C09128=1014.857,84.775,382.125,166.252,57.206,160.405
C09129=1014.862,85.025,382.109,166.255,57.195,160.404
C09130=1014.867,85.274,382.093,166.257,57.185,160.402
C09131=1014.871,85.523,382.077,166.260,57.175,160.401
C09132=1014.876,85.772,382.061,166.262,57.164,160.399
C09133=1014.881,86.022,382.045,166.265,57.155,160.398
C09134=1014.886,86.271,382.028,166.267,57.144,160.397
C09135=1014.890,86.521,382.013,166.270,57.133,160.395
C09136=1014.895,86.771,381.996,166.272,57.124,160.394
C09137=1014.899,87.020,381.980,166.275,57.113,160.392
C09138=1014.904,87.269,381.963,166.277,57.102,160.391
C09139=1014.909,87.518,381.948,166.280,57.093,160.390
C09140=1014.914,87.768,381.931,166.282,57.082,160.388
C09141=1014.919,88.018,381.916,166.285,57.071,160.387
C09142=1014.923,88.267,381.899,166.288,57.061,160.386
C09143=1014.928,88.517,381.883,166.290,57.051,160.384
C09144=1014.933,88.766,381.866,166.292,57.041,160.382
C09145=1014.937,89.015,381.850,166.296,57.031,160.381
C09146=1014.942,89.265,381.834,166.297,57.020,160.380
C09147=1014.946,89.514,381.817,166.301,57.010,160.378
C09148=1014.951,89.763,381.800,166.302,57.000,160.377
C09149=1014.956,90.013,381.783,166.306,56.990,160.376
C09150=1014.960,90.294,381.766,166.309,56.978,160.374
C09151=1014.966,90.575,381.747,166.311,56.967,160.372
C09152=1014.970,90.855,381.728,166.314,56.955,160.371
C09153=1014.976,91.135,381.710,166.317,56.944,160.369
C09154=1014.980,91.384,381.693,166.319,56.934,160.368
C09155=1014.985,91.634,381.676,166.323,56.924,160.367
C09156=1014.990,91.884,381.660,166.324,56.914,160.365
C09157=1014.994,92.133,381.644,166.327,56.903,160.364
C09158=1015.000,92.382,381.627,166.330,56.893,160.363
C09159=1015.003,92.631,381.610,166.332,56.883,160.361
C09160=1015.008,92.880,381.593,166.335,56.872,160.360
C09161=1015.013,93.131,381.577,166.338,56.862,160.358
C09162=1015.018,93.380,381.560,166.340,56.852,160.357
C09163=1015.022,93.630,381.543,166.343,56.841,160.355
C09164=1015.027,93.879,381.527,166.346,56.831,160.354
C09165=1015.031,94.128,381.510,166.348,56.821,160.353
C09166=1015.036,94.378,381.494,166.350,56.811,160.351
C09167=1015.041,94.627,381.477,166.354,56.801,160.350
C09168=1015.045,94.876,381.460,166.355,56.790,160.348
C09169=1015.050,95.126,381.444,166.358,56.780,160.347
C09170=1015.055,95.375,381.427,166.361,56.770,160.346
C09171=1015.060,95.624,381.410,166.364,56.759,160.344
C09172=1015.064,95.873,381.394,166.366,56.749,160.343
C09173=1015.069,96.124,381.377,166.369,56.738,160.341
C09174=1015.073,96.373,381.360,166.372,56.728,160.340
C09175=1015.078,96.622,381.344,166.375,56.718,160.339
C09176=1015.083,96.871,381.327,166.376,56.708,160.337
C09177=1015.087,97.121,381.310,166.379,56.697,160.336
C09178=1015.092,97.370,381.293,166.382,56.686,160.334
C09179=1015.097,97.619,381.277,166.385,56.676,160.333
C09180=1015.102,97.869,381.260,166.387,56.666,160.332
C09181=1015.106,98.118,381.243,166.390,56.656,160.330
C09182=1015.110,98.367,381.226,166.393,56.645,160.329
C09183=1015.115,98.618,381.210,166.395,56.634,160.327
C09184=1015.120,98.866,381.194,166.399,56.625,160.326
C09185=1015.124,99.116,381.176,166.401,56.614,160.325
C09186=1015.129,99.365,381.159,166.403,56.604,160.323
C09187=1015.134,99.615,381.142,166.407,56.594,160.322
C09188=1015.138,99.864,381.125,166.408,56.584,160.320
C09189=1015.143,100.114,381.108,166.411,56.573,160.319
C09190=1015.147,100.363,381.091,166.415,56.563,160.318
C09191=1015.152,100.613,381.074,166.416,56.553,160.316
C09192=1015.157,100.862,381.057,166.419,56.542,160.315
C09193=1015.161,101.112,381.040,166.422,56.532,160.313
C09194=1015.166,101.360,381.023,166.424,56.522,160.312
C09195=1015.170,101.610,381.005,166.427,56.512,160.311
C09196=1015.175,101.859,380.989,166.430,56.501,160.309
C09197=1015.179,102.109,380.971,166.433,56.491,160.308
C09198=1015.184,102.358,380.955,166.435,56.481,160.307
C09199=1015.189,102.608,380.937,166.438,56.471,160.305
C09200=1015.193,102.857,380.921,166.441,56.460,160.304
C09201=1015.198,103.106,380.903,166.444,56.449,160.302
C09202=1015.203,103.355,380.886,166.446,56.440,160.301
C09203=1015.207,103.605,380.869,166.449,56.429,160.300
C09204=1015.212,103.854,380.852,166.452,56.419,160.298
C09205=1015.216,104.104,380.835,166.455,56.408,160.297
C09206=1015.221,104.352,380.818,166.457,56.399,160.296
C09207=1015.226,104.602,380.800,166.460,56.388,160.294
C09208=1015.229,104.851,380.783,166.463,56.378,160.293
C09209=1015.235,105.101,380.766,166.466,56.367,160.291
C09210=1015.239,105.350,380.748,166.467,56.357,160.290
C09211=1015.244,105.599,380.732,166.470,56.346,160.288
C09212=1015.248,105.849,380.714,166.474,56.336,160.287
C09213=1015.253,106.098,380.698,166.477,56.326,160.286
C09214=1015.259,106.379,380.678,166.480,56.314,160.284
C09215=1015.263,106.660,380.658,166.482,56.302,160.282
C09216=1015.269,106.940,380.639,166.485,56.290,160.281
C09217=1015.275,107.222,380.620,166.488,56.279,160.279
C09218=1015.279,107.471,380.602,166.491,56.268,160.278
C09219=1015.284,107.720,380.585,166.494,56.258,160.277
C09220=1015.288,107.970,380.568,166.498,56.248,160.275
C09221=1015.293,108.219,380.551,166.500,56.238,160.274
C09222=1015.298,108.469,380.533,166.502,56.227,160.272
C09223=1015.302,108.717,380.517,166.505,56.217,160.271
C09224=1015.307,108.967,380.499,166.508,56.206,160.270
C09225=1015.311,109.216,380.482,166.511,56.196,160.268
C09226=1015.316,109.466,380.465,166.514,56.185,160.267
C09227=1015.321,109.715,380.447,166.516,56.175,160.265
C09228=1015.325,109.964,380.430,166.519,56.164,160.264
C09229=1015.330,110.213,380.412,166.522,56.155,160.263
C09230=1015.335,110.463,380.395,166.525,56.144,160.261
C09231=1015.339,110.713,380.377,166.528,56.133,160.260
C09232=1015.344,110.962,380.359,166.530,56.123,160.258
C09233=1015.348,111.211,380.343,166.533,56.113,160.257
C09234=1015.353,111.460,380.325,166.536,56.102,160.256
C09235=1015.357,111.710,380.307,166.539,56.092,160.254
C09236=1015.362,111.959,380.289,166.542,56.081,160.253
C09237=1015.366,112.209,380.272,166.544,56.072,160.252
C09238=1015.371,112.458,380.254,166.547,56.061,160.250
C09239=1015.375,112.707,380.236,166.550,56.051,160.249
C09240=1015.380,112.957,380.219,166.553,56.040,160.247
C09241=1015.384,113.206,380.200,166.556,56.031,160.246
C09242=1015.389,113.455,380.183,166.558,56.020,160.245
C09243=1015.393,113.705,380.165,166.561,56.010,160.243
C09244=1015.398,113.954,380.147,166.564,55.999,160.242
C09245=1015.402,114.203,380.129,166.567,55.990,160.241
C09246=1015.406,114.453,380.112,166.570,55.980,160.239
C09247=1015.411,114.702,380.094,166.573,55.969,160.238
C09248=1015.415,114.951,380.076,166.576,55.959,160.237
C09249=1015.420,115.201,380.058,166.578,55.949,160.235
C09250=1015.425,115.450,380.040,166.581,55.939,160.234
C09251=1015.429,115.700,380.022,166.584,55.928,160.232
C09252=1015.434,115.948,380.004,166.587,55.918,160.231
C09253=1015.438,116.198,379.987,166.590,55.907,160.230
C09254=1015.443,116.447,379.969,166.592,55.897,160.228
C09255=1015.447,116.696,379.951,166.596,55.887,160.227
C09256=1015.452,116.945,379.933,166.599,55.877,160.226
C09257=1015.456,117.195,379.915,166.602,55.866,160.224
C09258=1015.460,117.416,379.900,166.604,55.857,160.223
C09259=1015.464,117.636,379.883,166.607,55.848,160.222
C09260=1015.469,117.857,379.867,166.610,55.839,160.221
C09261=1015.473,118.078,379.852,166.611,55.830,160.219
C09262=1015.477,118.298,379.836,166.614,55.821,160.218
C09263=1015.481,118.519,379.821,166.617,55.812,160.217
C09264=1015.484,118.740,379.804,166.619,55.803,160.216
C09265=1015.488,118.961,379.788,166.622,55.793,160.214
C09266=1015.493,119.210,379.770,166.625,55.783,160.213
C09267=1015.497,119.459,379.753,166.628,55.773,160.212
C09268=1015.502,119.708,379.734,166.631,55.762,160.210
C09269=1015.507,119.957,379.716,166.634,55.752,160.209
C09270=1015.512,120.207,379.698,166.636,55.742,160.208
C09271=1015.516,120.456,379.681,166.639,55.732,160.206
C09272=1015.520,120.705,379.663,166.642,55.721,160.205
C09273=1015.525,120.955,379.645,166.645,55.711,160.204
C09274=1015.530,121.204,379.626,166.648,55.700,160.202
C09275=1015.535,121.453,379.608,166.651,55.690,160.201
C09276=1015.539,121.702,379.591,166.654,55.680,160.199
C09277=1015.543,121.952,379.573,166.657,55.669,160.198
C09278=1015.550,122.290,379.548,166.660,55.655,160.196
C09279=1015.556,122.628,379.524,166.665,55.641,160.194
C09280=1015.563,122.967,379.499,166.669,55.627,160.192
C09281=1015.568,123.305,379.475,166.674,55.613,160.191
C09282=1015.573,123.554,379.457,166.677,55.602,160.189
C09283=1015.578,123.804,379.439,166.680,55.592,160.188
C09284=1015.583,124.053,379.420,166.682,55.582,160.186
C09285=1015.588,124.302,379.402,166.685,55.571,160.185
C09286=1015.592,124.551,379.384,166.688,55.561,160.184
C09287=1015.597,124.800,379.366,166.691,55.551,160.182
C09288=1015.601,125.050,379.348,166.694,55.540,160.181
C09289=1015.606,125.299,379.330,166.697,55.530,160.180
C09290=1015.611,125.549,379.313,166.700,55.519,160.178
C09291=1015.615,125.798,379.294,166.703,55.509,160.177
C09292=1015.620,126.048,379.276,166.706,55.498,160.175
C09293=1015.625,126.297,379.258,166.709,55.487,160.174
C09294=1015.629,126.546,379.240,166.712,55.477,160.173
C09295=1015.634,126.795,379.222,166.715,55.466,160.171
C09296=1015.639,127.044,379.204,166.718,55.456,160.170
C09297=1015.643,127.294,379.186,166.722,55.446,160.168
C09298=1015.648,127.543,379.168,166.725,55.435,160.167
C09299=1015.653,127.792,379.149,166.728,55.425,160.166
C09300=1015.658,128.042,379.131,166.731,55.414,160.164
C09301=1015.663,128.291,379.113,166.734,55.404,160.163
C09302=1015.667,128.540,379.095,166.737,55.394,160.162
C09303=1015.671,128.790,379.076,166.740,55.383,160.160
C09304=1015.676,129.039,379.057,166.743,55.372,160.159
C09305=1015.681,129.288,379.039,166.746,55.362,160.157
C09306=1015.685,129.537,379.021,166.749,55.351,160.156
C09307=1015.690,129.786,379.003,166.752,55.341,160.155
C09308=1015.694,130.036,378.984,166.755,55.330,160.153
C09309=1015.700,130.286,378.966,166.758,55.320,160.152
C09310=1015.704,130.535,378.948,166.762,55.310,160.151
C09311=1015.708,130.784,378.929,166.765,55.300,160.149
C09312=1015.713,131.033,378.911,166.768,55.290,160.148
C09313=1015.717,131.283,378.892,166.772,55.279,160.147
C09314=1015.722,131.531,378.873,166.775,55.269,160.145
C09315=1015.727,131.781,378.855,166.777,55.259,160.144
C09316=1015.731,132.030,378.836,166.780,55.249,160.143
C09317=1015.736,132.280,378.818,166.783,55.238,160.141
C09318=1015.740,132.529,378.798,166.786,55.228,160.140
C09319=1015.745,132.778,378.780,166.789,55.217,160.138
C09320=1015.750,133.027,378.762,166.793,55.207,160.137
C09321=1015.754,133.276,378.743,166.796,55.197,160.136
C09322=1015.759,133.526,378.724,166.799,55.186,160.134
C09323=1015.763,133.775,378.706,166.802,55.176,160.133
C09324=1015.768,134.024,378.687,166.805,55.166,160.132
C09325=1015.773,134.274,378.669,166.808,55.155,160.130
C09326=1015.777,134.523,378.650,166.812,55.145,160.129
C09327=1015.782,134.772,378.631,166.815,55.135,160.128
C09328=1015.786,135.021,378.613,166.818,55.124,160.126
C09329=1015.791,135.270,378.593,166.821,55.114,160.125
C09330=1015.796,135.520,378.575,166.824,55.103,160.124
C09331=1015.800,135.769,378.556,166.828,55.093,160.122
C09332=1015.805,136.018,378.538,166.831,55.083,160.121
C09333=1015.809,136.268,378.519,166.834,55.072,160.120
C09334=1015.814,136.516,378.500,166.837,55.062,160.118
C09335=1015.818,136.766,378.481,166.840,55.052,160.117
C09336=1015.823,137.015,378.462,166.844,55.041,160.116
C09337=1015.828,137.265,378.443,166.847,55.031,160.114
C09338=1015.833,137.514,378.424,166.850,55.021,160.113
C09339=1015.837,137.764,378.406,166.853,55.010,160.112
C09340=1015.842,138.012,378.387,166.856,55.000,160.110
C09341=1015.846,138.262,378.368,166.860,54.990,160.109
C09342=1015.851,138.543,378.346,166.863,54.978,160.107
C09343=1015.856,138.823,378.325,166.867,54.967,160.106
C09344=1015.861,139.104,378.304,166.871,54.955,160.105
C09345=1015.866,139.385,378.282,166.874,54.943,160.103
C09346=1015.871,139.634,378.263,166.877,54.933,160.102
C09347=1015.875,139.884,378.244,166.881,54.923,160.100
C09348=1015.879,140.133,378.225,166.884,54.913,160.099
C09349=1015.885,140.382,378.205,166.888,54.903,160.098
C09350=1015.889,140.632,378.187,166.891,54.892,160.096
C09351=1015.894,140.881,378.167,166.894,54.882,160.095
C09352=1015.899,141.129,378.148,166.897,54.872,160.094
C09353=1015.903,141.379,378.130,166.901,54.861,160.092
C09354=1015.907,141.628,378.110,166.904,54.851,160.091
C09355=1015.912,141.877,378.091,166.907,54.841,160.090
C09356=1015.916,142.127,378.072,166.910,54.831,160.088
C09357=1015.921,142.376,378.053,166.914,54.820,160.087
C09358=1015.926,142.625,378.034,166.917,54.810,160.086
C09359=1015.930,142.875,378.015,166.920,54.800,160.084
C09360=1015.935,143.123,377.996,166.923,54.789,160.083
C09361=1015.940,143.373,377.977,166.927,54.779,160.082
C09362=1015.944,143.622,377.957,166.930,54.769,160.080
C09363=1015.949,143.872,377.939,166.933,54.759,160.079
C09364=1015.954,144.121,377.919,166.937,54.748,160.078
C09365=1015.958,144.370,377.900,166.940,54.738,160.076
C09366=1015.963,144.618,377.881,166.943,54.728,160.075
C09367=1015.967,144.868,377.862,166.946,54.717,160.074
C09368=1015.972,145.117,377.843,166.950,54.707,160.072
C09369=1015.977,145.367,377.823,166.953,54.697,160.071
C09370=1015.982,145.616,377.804,166.956,54.687,160.070
C09371=1015.986,145.865,377.784,166.960,54.676,160.068
C09372=1015.990,146.114,377.765,166.963,54.666,160.067
C09373=1015.995,146.363,377.745,166.966,54.656,160.066
C09374=1015.999,146.613,377.726,166.970,54.645,160.064
C09375=1016.004,146.862,377.707,166.973,54.635,160.063
C09376=1016.008,147.111,377.687,166.976,54.625,160.062
C09377=1016.013,147.360,377.669,166.979,54.615,160.061
C09378=1016.018,147.610,377.649,166.984,54.604,160.059
C09379=1016.022,147.859,377.629,166.987,54.594,160.058
C09380=1016.027,148.108,377.610,166.990,54.583,160.057
C09381=1016.031,148.357,377.590,166.994,54.573,160.055
C09382=1016.036,148.607,377.570,166.997,54.563,160.054
C09383=1016.040,148.856,377.551,167.000,54.553,160.053
C09384=1016.045,149.105,377.531,167.004,54.543,160.052
C09385=1016.049,149.354,377.512,167.008,54.533,160.050
C09386=1016.054,149.603,377.492,167.011,54.523,160.049
C09387=1016.058,149.852,377.473,167.014,54.512,160.048
C09388=1016.063,150.101,377.453,167.018,54.502,160.046
C09389=1016.068,150.351,377.433,167.021,54.492,160.045
C09390=1016.072,150.600,377.414,167.024,54.482,160.044
C09391=1016.077,150.849,377.395,167.028,54.472,160.042
C09392=1016.082,151.097,377.375,167.031,54.461,160.041
C09393=1016.087,151.347,377.355,167.034,54.451,160.040
C09394=1016.091,151.596,377.336,167.038,54.441,160.038
C09395=1016.095,151.845,377.316,167.041,54.431,160.037
C09396=1016.100,152.095,377.296,167.045,54.420,160.036
C09397=1016.105,152.344,377.277,167.049,54.410,160.035
C09398=1016.109,152.593,377.257,167.052,54.400,160.033
C09399=1016.114,152.843,377.237,167.056,54.389,160.032
C09400=1016.119,153.091,377.217,167.059,54.379,160.031
C09401=1016.123,153.340,377.198,167.062,54.369,160.029
C09402=1016.127,153.590,377.177,167.066,54.359,160.028
C09403=1016.132,153.839,377.158,167.070,54.349,160.027
C09404=1016.136,154.088,377.138,167.073,54.339,160.026
C09405=1016.141,154.338,377.118,167.076,54.329,160.024
C09406=1016.146,154.618,377.096,167.080,54.317,160.023
C09407=1016.152,154.899,377.073,167.084,54.305,160.021
C09408=1016.157,155.180,377.051,167.089,54.294,160.020
C09409=1016.162,155.460,377.029,167.093,54.282,160.019
C09410=1016.166,155.710,377.008,167.096,54.272,160.017
C09411=1016.171,155.959,376.989,167.099,54.262,160.016
C09412=1016.176,156.209,376.969,167.103,54.252,160.015
C09413=1016.180,156.457,376.949,167.106,54.242,160.013
C09414=1016.185,156.706,376.929,167.110,54.231,160.012
C09415=1016.189,156.956,376.909,167.113,54.221,160.011
C09416=1016.194,157.204,376.889,167.118,54.211,160.010
C09417=1016.199,157.454,376.869,167.121,54.201,160.008
C09418=1016.203,157.703,376.850,167.125,54.191,160.007
C09419=1016.207,157.952,376.829,167.128,54.181,160.006
C09420=1016.212,158.202,376.809,167.132,54.171,160.004
C09421=1016.217,158.451,376.790,167.135,54.160,160.003
C09422=1016.222,158.700,376.769,167.139,54.150,160.002
C09423=1016.226,158.948,376.749,167.142,54.140,160.001
C09424=1016.231,159.198,376.729,167.146,54.131,159.999
C09425=1016.235,159.447,376.708,167.149,54.121,159.998
C09426=1016.238,159.696,376.688,167.153,54.110,159.997
C09427=1016.244,159.945,376.667,167.157,54.101,159.996
C09428=1016.247,160.194,376.646,167.160,54.091,159.994
C09429=1016.252,160.444,376.627,167.164,54.081,159.993
C09430=1016.256,160.693,376.606,167.167,54.070,159.992
C09431=1016.261,160.942,376.585,167.171,54.061,159.991
C09432=1016.265,161.191,376.565,167.174,54.051,159.990
C09433=1016.270,161.441,376.544,167.178,54.041,159.988
C09434=1016.274,161.689,376.524,167.181,54.030,159.987
C09435=1016.279,161.938,376.503,167.185,54.021,159.986
C09436=1016.283,162.187,376.483,167.190,54.010,159.985
C09437=1016.287,162.436,376.463,167.193,54.000,159.983
C09438=1016.292,162.686,376.441,167.197,53.991,159.982
C09439=1016.296,162.935,376.422,167.201,53.981,159.981
C09440=1016.301,163.184,376.401,167.204,53.971,159.980
C09441=1016.306,163.433,376.380,167.208,53.960,159.978
C09442=1016.310,163.682,376.359,167.211,53.951,159.977
C09443=1016.314,163.932,376.339,167.215,53.941,159.976
C09444=1016.319,164.180,376.319,167.218,53.931,159.975
C09445=1016.323,164.430,376.298,167.222,53.921,159.973
C09446=1016.328,164.678,376.277,167.226,53.911,159.972
C09447=1016.332,164.928,376.256,167.229,53.901,159.971
C09448=1016.337,165.177,376.237,167.234,53.891,159.970
C09449=1016.341,165.426,376.216,167.237,53.880,159.969
C09450=1016.345,165.675,376.195,167.241,53.870,159.967
C09451=1016.350,165.924,376.174,167.245,53.861,159.966
C09452=1016.354,166.173,376.154,167.248,53.851,159.965
C09453=1016.359,166.422,376.133,167.252,53.841,159.964
C09454=1016.364,166.672,376.113,167.255,53.831,159.962
C09455=1016.368,166.921,376.092,167.259,53.821,159.961
C09456=1016.373,167.170,376.071,167.264,53.811,159.960
C09457=1016.377,167.419,376.050,167.267,53.801,159.959
C09458=1016.382,167.668,376.030,167.271,53.790,159.957
C09459=1016.387,167.917,376.009,167.274,53.780,159.956
C09460=1016.390,168.166,375.988,167.278,53.771,159.955
C09461=1016.396,168.415,375.967,167.282,53.761,159.954
C09462=1016.400,168.664,375.946,167.286,53.750,159.953
C09463=1016.405,168.913,375.926,167.290,53.740,159.951
C09464=1016.409,169.163,375.906,167.294,53.730,159.950
C09465=1016.413,169.412,375.885,167.298,53.721,159.949
C09466=1016.418,169.661,375.864,167.301,53.711,159.948
C09467=1016.423,169.910,375.843,167.306,53.700,159.947
C09468=1016.427,170.159,375.823,167.309,53.690,159.945
C09469=1016.432,170.408,375.802,167.313,53.680,159.944
C09470=1016.437,170.688,375.778,167.317,53.669,159.943
C09471=1016.443,170.969,375.755,167.321,53.658,159.941
C09472=1016.447,171.250,375.732,167.326,53.646,159.940
C09473=1016.453,171.530,375.707,167.330,53.635,159.938
C09474=1016.458,171.779,375.687,167.334,53.625,159.937
C09475=1016.462,172.028,375.666,167.339,53.615,159.936
C09476=1016.467,172.277,375.645,167.342,53.605,159.935
C09477=1016.472,172.527,375.624,167.346,53.595,159.934
C09478=1016.476,172.775,375.603,167.349,53.585,159.932
C09479=1016.481,173.024,375.583,167.354,53.575,159.931
C09480=1016.486,173.274,375.562,167.358,53.564,159.930
C09481=1016.490,173.522,375.542,167.362,53.555,159.929
C09482=1016.495,173.772,375.520,167.365,53.545,159.928
C09483=1016.499,174.021,375.499,167.370,53.535,159.926
C09484=1016.505,174.270,375.479,167.373,53.525,159.925
C09485=1016.509,174.520,375.458,167.377,53.515,159.924
C09486=1016.513,174.769,375.437,167.382,53.505,159.923
C09487=1016.519,175.017,375.416,167.386,53.495,159.922
C09488=1016.523,175.266,375.394,167.389,53.485,159.920
C09489=1016.528,175.516,375.374,167.393,53.475,159.919
C09490=1016.532,175.764,375.353,167.397,53.464,159.918
C09491=1016.537,176.014,375.332,167.401,53.454,159.917
C09492=1016.542,176.263,375.311,167.405,53.444,159.915
C09493=1016.547,176.512,375.289,167.410,53.434,159.914
C09494=1016.552,176.761,375.269,167.413,53.424,159.913
C09495=1016.557,177.010,375.248,167.417,53.414,159.912
C09496=1016.561,177.259,375.227,167.422,53.404,159.911
C09497=1016.566,177.508,375.206,167.425,53.394,159.909
C09498=1016.571,177.757,375.185,167.429,53.384,159.908
C09499=1016.576,178.006,375.164,167.434,53.374,159.907
C09500=1016.580,178.255,375.143,167.438,53.364,159.906
C09501=1016.585,178.505,375.122,167.442,53.354,159.905
C09502=1016.590,178.753,375.100,167.446,53.344,159.903
C09503=1016.594,179.002,375.080,167.449,53.334,159.902
C09504=1016.599,179.252,375.059,167.454,53.323,159.901
C09505=1016.604,179.501,375.038,167.458,53.313,159.900
C09506=1016.609,179.750,375.016,167.462,53.304,159.899
C09507=1016.614,179.999,374.996,167.466,53.294,159.897
C09508=1016.619,180.248,374.974,167.470,53.284,159.896
C09509=1016.624,180.497,374.953,167.475,53.273,159.895
C09510=1016.629,180.746,374.932,167.478,53.263,159.894
C09511=1016.633,180.995,374.911,167.482,53.253,159.892
C09512=1016.638,181.244,374.889,167.487,53.244,159.891
C09513=1016.643,181.493,374.868,167.491,53.234,159.890
C09514=1016.648,181.742,374.847,167.495,53.223,159.889
C09515=1016.653,181.992,374.825,167.499,53.213,159.888
C09516=1016.658,182.240,374.804,167.503,53.204,159.887
C09517=1016.661,182.490,374.782,167.507,53.194,159.885
C09518=1016.666,182.738,374.760,167.512,53.184,159.884
C09519=1016.670,182.987,374.738,167.516,53.174,159.883
C09520=1016.674,183.237,374.717,167.520,53.165,159.882
C09521=1016.679,183.486,374.695,167.523,53.155,159.881
C09522=1016.684,183.735,374.673,167.529,53.145,159.880
C09523=1016.689,183.983,374.651,167.532,53.135,159.879
C09524=1016.693,184.232,374.629,167.536,53.126,159.878
C09525=1016.697,184.482,374.607,167.540,53.116,159.876
C09526=1016.702,184.731,374.586,167.545,53.106,159.875
C09527=1016.707,184.980,374.564,167.549,53.097,159.874
C09528=1016.711,185.229,374.541,167.553,53.087,159.873
C09529=1016.716,185.477,374.519,167.557,53.077,159.872
C09530=1016.720,185.727,374.498,167.561,53.067,159.871
C09531=1016.724,185.976,374.476,167.566,53.058,159.869
C09532=1016.729,186.225,374.454,167.569,53.048,159.868
C09533=1016.734,186.474,374.432,167.574,53.038,159.867
C09534=1016.739,186.754,374.408,167.579,53.027,159.866
C09535=1016.744,187.034,374.382,167.583,53.016,159.865
C09536=1016.750,187.315,374.358,167.589,53.005,159.863
C09537=1016.754,187.594,374.333,167.593,52.994,159.862
C09538=1016.759,187.844,374.312,167.597,52.984,159.861
C09539=1016.764,188.093,374.290,167.602,52.975,159.860
C09540=1016.768,188.341,374.268,167.606,52.965,159.859
C09541=1016.772,188.590,374.246,167.610,52.956,159.858
C09542=1016.778,188.840,374.223,167.614,52.945,159.856
C09543=1016.783,189.089,374.201,167.619,52.936,159.855
C09544=1016.787,189.338,374.180,167.623,52.926,159.854
C09545=1016.792,189.587,374.157,167.628,52.916,159.853
C09546=1016.796,189.836,374.135,167.631,52.907,159.852
C09547=1016.801,190.084,374.113,167.636,52.897,159.851
C09548=1016.805,190.333,374.091,167.640,52.887,159.850
C09549=1016.810,190.582,374.069,167.644,52.878,159.849
C09550=1016.815,190.831,374.047,167.649,52.867,159.847
C09551=1016.820,191.080,374.025,167.653,52.858,159.846
C09552=1016.824,191.330,374.003,167.658,52.848,159.845
C09553=1016.829,191.579,373.981,167.662,52.839,159.844
C09554=1016.834,191.827,373.959,167.666,52.829,159.843
C09555=1016.838,192.077,373.936,167.671,52.819,159.842
C09556=1016.843,192.325,373.914,167.675,52.809,159.841
C09557=1016.848,192.574,373.893,167.680,52.799,159.840
C09558=1016.854,192.823,373.870,167.684,52.790,159.838
C09559=1016.858,193.072,373.847,167.689,52.780,159.837
C09560=1016.862,193.321,373.825,167.693,52.770,159.836
C09561=1016.867,193.570,373.803,167.698,52.760,159.835
C09562=1016.871,193.819,373.781,167.702,52.751,159.834
C09563=1016.877,194.068,373.759,167.706,52.741,159.833
C09564=1016.882,194.317,373.737,167.711,52.731,159.832
C09565=1016.886,194.566,373.714,167.715,52.722,159.831
C09566=1016.891,194.815,373.692,167.720,52.712,159.830
C09567=1016.896,195.063,373.670,167.724,52.702,159.828
C09568=1016.901,195.313,373.648,167.729,52.693,159.827
C09569=1016.905,195.562,373.625,167.733,52.683,159.826
C09570=1016.910,195.811,373.603,167.738,52.673,159.825
C09571=1016.915,196.059,373.581,167.742,52.663,159.824
C09572=1016.920,196.309,373.558,167.747,52.654,159.823
C09573=1016.925,196.558,373.536,167.751,52.644,159.822
C09574=1016.929,196.806,373.514,167.756,52.634,159.821
C09575=1016.934,197.056,373.491,167.760,52.624,159.819
C09576=1016.939,197.305,373.469,167.765,52.615,159.819
C09577=1016.944,197.553,373.447,167.769,52.605,159.817
C09578=1016.950,197.802,373.424,167.774,52.595,159.816
C09579=1016.954,198.051,373.402,167.779,52.585,159.815
C09580=1016.959,198.300,373.380,167.783,52.576,159.814
C09581=1016.964,198.549,373.357,167.788,52.566,159.813
C09582=1016.969,198.798,373.334,167.792,52.556,159.812
C09583=1016.973,199.047,373.313,167.797,52.546,159.811
C09584=1016.979,199.296,373.290,167.801,52.537,159.810
C09585=1016.983,199.545,373.267,167.806,52.527,159.809
C09586=1016.988,199.794,373.244,167.810,52.518,159.808
C09587=1016.992,200.043,373.221,167.816,52.508,159.807
C09588=1016.997,200.292,373.199,167.819,52.499,159.805
C09589=1017.002,200.541,373.176,167.825,52.489,159.804
C09590=1017.006,200.790,373.153,167.829,52.480,159.803
C09591=1017.012,201.038,373.130,167.834,52.470,159.802
C09592=1017.016,201.287,373.108,167.838,52.460,159.801
C09593=1017.021,201.536,373.084,167.843,52.451,159.800
C09594=1017.026,201.785,373.061,167.847,52.441,159.799
C09595=1017.030,202.033,373.038,167.852,52.432,159.798
C09596=1017.035,202.281,373.016,167.857,52.423,159.797
C09597=1017.058,203.524,372.902,168.348,52.501,159.911
C09598=1017.064,203.761,372.878,168.352,52.493,159.910
C09599=1017.070,203.999,372.855,168.356,52.485,159.909
C09600=1017.075,204.236,372.832,168.359,52.477,159.908
C09601=1017.081,204.474,372.808,168.364,52.469,159.907
C09602=1017.086,204.712,372.785,168.368,52.461,159.906
C09603=1017.092,204.949,372.761,168.371,52.453,159.905
C09604=1017.097,205.187,372.737,168.375,52.445,159.904
C09605=1017.103,205.425,372.714,168.379,52.437,159.903
C09606=1017.109,205.673,372.689,168.383,52.429,159.902
C09607=1017.114,205.922,372.665,168.387,52.421,159.901
C09608=1017.120,206.171,372.640,168.390,52.413,159.900
C09609=1017.126,206.419,372.615,168.395,52.404,159.899
C09610=1017.132,206.668,372.590,168.399,52.396,159.898
C09611=1017.138,206.916,372.566,168.403,52.387,159.897
C09612=1017.144,207.165,372.541,168.407,52.379,159.896
C09613=1017.149,207.413,372.516,168.411,52.371,159.895
C09614=1017.155,207.663,372.491,168.415,52.362,159.894
C09615=1017.160,207.912,372.467,168.418,52.354,159.893
C09616=1017.166,208.160,372.442,168.423,52.346,159.892
C09617=1017.172,208.409,372.417,168.427,52.338,159.891
C09618=1017.178,208.657,372.392,168.431,52.330,159.890
C09619=1017.183,208.907,372.367,168.435,52.322,159.889
C09620=1017.189,209.155,372.342,168.439,52.314,159.888
C09621=1017.195,209.404,372.318,168.444,52.306,159.888
C09622=1017.201,209.653,372.292,168.447,52.298,159.887
C09623=1017.207,209.901,372.268,168.451,52.290,159.886
C09624=1017.212,210.150,372.242,168.456,52.281,159.885
C09625=1017.218,210.398,372.217,168.459,52.273,159.884
C09626=1017.224,210.647,372.192,168.463,52.265,159.883
C09627=1017.230,210.896,372.167,168.468,52.258,159.882
C09628=1017.235,211.144,372.142,168.472,52.250,159.881
C09629=1017.241,211.393,372.116,168.475,52.242,159.880
C09630=1017.246,211.642,372.092,168.479,52.234,159.879
C09631=1017.252,211.890,372.067,168.484,52.226,159.878
C09632=1017.258,212.139,372.041,168.488,52.218,159.877
C09633=1017.263,212.388,372.017,168.491,52.210,159.876
C09634=1017.269,212.636,371.991,168.496,52.202,159.875
C09635=1017.275,212.885,371.966,168.500,52.194,159.875
C09636=1017.280,213.133,371.940,168.504,52.186,159.874
C09637=1017.286,213.383,371.916,168.507,52.178,159.873
C09638=1017.292,213.631,371.890,168.513,52.171,159.872
C09639=1017.298,213.879,371.866,168.516,52.163,159.871
C09640=1017.303,214.128,371.840,168.520,52.155,159.870
C09641=1017.310,214.377,371.814,168.524,52.147,159.869
C09642=1017.316,214.626,371.790,168.529,52.139,159.868
C09643=1017.321,214.874,371.765,168.533,52.132,159.867
C09644=1017.327,215.123,371.739,168.536,52.124,159.866
C09645=1017.333,215.372,371.713,168.540,52.116,159.865
C09646=1017.338,215.620,371.688,168.545,52.108,159.865
C09647=1017.345,215.869,371.663,168.549,52.100,159.864
C09648=1017.350,216.118,371.638,168.553,52.093,159.863
C09649=1017.356,216.367,371.613,168.557,52.085,159.862
C09650=1017.362,216.615,371.588,168.562,52.077,159.861
C09651=1017.367,216.864,371.562,168.565,52.069,159.860
C09652=1017.373,217.112,371.536,168.570,52.062,159.859
C09653=1017.379,217.361,371.511,168.573,52.054,159.858
C09654=1017.385,217.609,371.486,168.578,52.046,159.858
C09655=1017.391,217.858,371.460,168.582,52.038,159.857
C09656=1017.397,218.107,371.435,168.586,52.031,159.856
C09657=1017.403,218.355,371.409,168.590,52.023,159.855
C09658=1017.408,218.590,371.385,168.594,52.016,159.854
C09659=1017.414,218.824,371.361,168.598,52.008,159.853
C09660=1017.419,219.059,371.337,168.602,52.002,159.853
C09661=1017.424,219.294,371.313,168.606,51.995,159.852
C09662=1017.429,219.528,371.288,168.610,51.987,159.851
C09663=1017.434,219.763,371.263,168.613,51.980,159.850
C09664=1017.440,219.998,371.240,168.617,51.973,159.849
C09665=1017.445,220.233,371.215,168.621,51.966,159.849
C09666=1017.451,220.481,371.190,168.625,51.959,159.848
C09667=1017.457,220.729,371.163,168.629,51.951,159.847
C09668=1017.463,220.978,371.138,168.634,51.944,159.846
C09669=1017.469,221.227,371.112,168.637,51.936,159.845
C09670=1017.475,221.476,371.087,168.641,51.929,159.844
C09671=1017.480,221.724,371.061,168.647,51.921,159.844
C09672=1017.487,221.973,371.035,168.651,51.914,159.843
C09673=1017.492,222.221,371.009,168.655,51.907,159.842
C09674=1017.497,222.470,370.983,168.659,51.899,159.841
C09675=1017.503,222.718,370.958,168.663,51.891,159.840
C09676=1017.509,222.967,370.931,168.667,51.884,159.840
C09677=1017.515,223.215,370.906,168.671,51.877,159.839
C09678=1017.521,223.464,370.880,168.675,51.870,159.838
C09679=1017.527,223.713,370.855,168.679,51.862,159.837
C09680=1017.533,223.961,370.828,168.683,51.855,159.836
C09681=1017.538,224.210,370.802,168.687,51.848,159.836
C09682=1017.544,224.459,370.777,168.692,51.841,159.835
C09683=1017.550,224.708,370.750,168.697,51.833,159.834
C09684=1017.556,224.956,370.725,168.701,51.826,159.833
C09685=1017.561,225.204,370.699,168.705,51.818,159.833
C09686=1017.567,225.453,370.673,168.709,51.811,159.831
C09687=1017.573,225.701,370.647,168.713,51.803,159.831
C09688=1017.579,225.950,370.621,168.717,51.796,159.830
C09689=1017.585,226.199,370.595,168.721,51.789,159.829
C09690=1017.591,226.447,370.569,168.725,51.782,159.828
C09691=1017.596,226.696,370.543,168.730,51.775,159.828
C09692=1017.603,226.944,370.517,168.734,51.768,159.827
C09693=1017.608,227.193,370.491,168.738,51.760,159.826
C09694=1017.614,227.441,370.464,168.742,51.753,159.825
C09695=1017.620,227.690,370.438,168.747,51.746,159.825
C09696=1017.625,227.939,370.411,168.751,51.739,159.824
C09697=1017.631,228.188,370.386,168.755,51.732,159.823
C09698=1017.637,228.436,370.359,168.759,51.725,159.822
C09699=1017.643,228.684,370.333,168.764,51.718,159.822
C09700=1017.649,228.933,370.307,168.768,51.710,159.821
C09701=1017.654,229.181,370.280,168.772,51.704,159.820
C09702=1017.660,229.430,370.254,168.776,51.697,159.819
C09703=1017.666,229.679,370.228,168.781,51.689,159.819
C09704=1017.672,229.927,370.202,168.785,51.682,159.818
C09705=1017.678,230.175,370.175,168.788,51.676,159.817
C09706=1017.683,230.424,370.149,168.793,51.669,159.816
C09707=1017.690,230.673,370.122,168.797,51.662,159.816
C09708=1017.696,230.921,370.095,168.801,51.655,159.815
C09709=1017.701,231.170,370.069,168.805,51.648,159.814
C09710=1017.707,231.419,370.043,168.810,51.641,159.814
C09711=1017.713,231.667,370.016,168.814,51.634,159.813
C09712=1017.718,231.916,369.990,168.818,51.627,159.812
C09713=1017.724,232.164,369.963,168.823,51.620,159.812
C09714=1017.730,232.412,369.936,168.827,51.613,159.811
C09715=1017.736,232.661,369.910,168.832,51.606,159.810
C09716=1017.741,232.910,369.884,168.835,51.600,159.809
C09717=1017.747,233.159,369.857,168.840,51.593,159.809
C09718=1017.752,233.389,369.832,168.844,51.586,159.808
C09719=1017.758,233.619,369.807,168.848,51.580,159.807
C09720=1017.764,233.850,369.783,168.851,51.574,159.807
C09721=1017.769,234.080,369.758,168.856,51.568,159.806
C09722=1017.774,234.310,369.733,168.859,51.561,159.805
C09723=1017.780,234.542,369.709,168.864,51.555,159.805
C09724=1017.785,234.772,369.684,168.868,51.549,159.804
C09725=1017.790,235.002,369.659,168.871,51.543,159.804
C09726=1017.797,235.251,369.632,168.875,51.535,159.803
C09727=1017.802,235.499,369.605,168.880,51.529,159.802
C09728=1017.808,235.748,369.579,168.884,51.522,159.801
C09729=1017.814,235.996,369.552,168.889,51.515,159.801
C09730=1017.820,236.244,369.525,168.893,51.509,159.800
C09731=1017.826,236.493,369.498,168.898,51.501,159.799
C09732=1017.832,236.742,369.472,168.901,51.495,159.799
C09733=1017.838,236.990,369.445,168.906,51.489,159.798
C09734=1017.843,237.238,369.418,168.910,51.481,159.797
C09735=1017.850,237.488,369.391,168.915,51.475,159.797
C09736=1017.856,237.736,369.365,168.919,51.468,159.796
C09737=1017.861,237.984,369.338,168.923,51.461,159.795
C09738=1017.867,238.232,369.311,168.928,51.455,159.795
C09739=1017.873,238.480,369.284,168.932,51.449,159.794
C09740=1017.880,238.729,369.257,168.936,51.442,159.794
C09741=1017.885,238.978,369.230,168.940,51.435,159.793
C09742=1017.890,239.226,369.203,168.945,51.428,159.792
C09743=1017.896,239.474,369.176,168.950,51.422,159.792
C09744=1017.903,239.723,369.149,168.953,51.416,159.791
C09745=1017.908,239.972,369.121,168.958,51.409,159.790
C09746=1017.914,240.220,369.094,168.963,51.403,159.790
C09747=1017.920,240.469,369.067,168.967,51.396,159.789
C09748=1017.925,240.717,369.040,168.971,51.390,159.788
C09749=1017.931,240.965,369.013,168.975,51.383,159.788
C09750=1017.937,241.213,368.986,168.980,51.377,159.787
C09751=1017.943,241.463,368.958,168.985,51.370,159.787
C09752=1017.949,241.711,368.931,168.988,51.364,159.786
C09753=1017.955,241.959,368.904,168.993,51.358,159.785
C09754=1017.961,242.208,368.876,168.997,51.351,159.785
C09755=1017.966,242.456,368.849,169.002,51.345,159.784
C09756=1017.972,242.704,368.823,169.006,51.339,159.784
C09757=1017.978,242.953,368.794,169.010,51.332,159.783
C09758=1017.984,243.202,368.768,169.015,51.326,159.782
C09759=1017.989,243.450,368.740,169.020,51.319,159.782
C09760=1017.996,243.699,368.713,169.023,51.313,159.781
C09761=1018.001,243.947,368.685,169.028,51.307,159.781
C09762=1018.007,244.195,368.656,169.033,51.301,159.780
C09763=1018.013,244.444,368.630,169.036,51.295,159.780
C09764=1018.018,244.692,368.602,169.041,51.288,159.779
C09765=1018.025,244.940,368.574,169.046,51.282,159.778
C09766=1018.030,245.189,368.547,169.050,51.276,159.778
C09767=1018.035,245.437,368.519,169.054,51.270,159.777
C09768=1018.042,245.685,368.491,169.059,51.263,159.777
C09769=1018.047,245.934,368.464,169.063,51.257,159.776
C09770=1018.053,246.183,368.436,169.068,51.251,159.776
C09771=1018.059,246.431,368.408,169.072,51.245,159.775
C09772=1018.064,246.680,368.381,169.076,51.239,159.774
C09773=1018.070,246.928,368.353,169.081,51.233,159.774
C09774=1018.076,247.176,368.325,169.086,51.226,159.773
C09775=1018.082,247.425,368.297,169.089,51.220,159.773
C09776=1018.088,247.672,368.270,169.094,51.214,159.772
C09777=1018.093,247.922,368.242,169.099,51.208,159.772
C09778=1018.099,248.148,368.216,169.103,51.203,159.771
C09779=1018.104,248.376,368.191,169.107,51.197,159.771
C09780=1018.110,248.603,368.165,169.111,51.192,159.770
C09781=1018.115,248.830,368.141,169.115,51.186,159.770
C09782=1018.121,249.057,368.115,169.119,51.181,159.769
C09783=1018.126,249.284,368.090,169.123,51.175,159.769
C09784=1018.131,249.511,368.064,169.127,51.169,159.768
C09785=1018.137,249.739,368.038,169.131,51.164,159.768
C09786=1018.142,249.987,368.010,169.136,51.158,159.767
C09787=1018.149,250.236,367.983,169.141,51.151,159.767
C09788=1018.154,250.484,367.955,169.145,51.146,159.766
C09789=1018.160,250.733,367.927,169.149,51.140,159.766
C09790=1018.166,250.980,367.899,169.153,51.134,159.765
C09791=1018.172,251.229,367.871,169.158,51.128,159.765
C09792=1018.179,251.478,367.843,169.163,51.122,159.764
C09793=1018.184,251.726,367.815,169.167,51.116,159.764
C09794=1018.190,251.974,367.787,169.172,51.110,159.763
C09795=1018.196,252.222,367.760,169.176,51.104,159.763
C09796=1018.202,252.471,367.731,169.180,51.098,159.762
C09797=1018.208,252.720,367.703,169.185,51.092,159.762
C09798=1018.214,252.967,367.676,169.190,51.086,159.761
C09799=1018.220,253.216,367.647,169.194,51.080,159.761
C09800=1018.226,253.465,367.619,169.199,51.074,159.760
C09801=1018.232,253.713,367.592,169.204,51.068,159.760
C09802=1018.238,253.961,367.563,169.208,51.063,159.759
C09803=1018.244,254.210,367.536,169.213,51.056,159.759
C09804=1018.250,254.458,367.508,169.217,51.051,159.758
C09805=1018.256,254.707,367.479,169.222,51.045,159.758
C09806=1018.263,254.954,367.451,169.226,51.039,159.757
C09807=1018.268,255.202,367.423,169.230,51.033,159.757
C09808=1018.274,255.451,367.395,169.235,51.027,159.756
C09809=1018.281,255.700,367.367,169.240,51.021,159.756
C09810=1018.286,255.948,367.339,169.244,51.016,159.755
C09811=1018.292,256.196,367.311,169.249,51.010,159.755
C09812=1018.299,256.445,367.283,169.254,51.004,159.755
C09813=1018.305,256.693,367.254,169.258,50.998,159.754
C09814=1018.310,256.941,367.226,169.263,50.992,159.754
C09815=1018.317,257.190,367.198,169.267,50.987,159.753
C09816=1018.323,257.438,367.170,169.272,50.981,159.753
C09817=1018.329,257.686,367.141,169.277,50.975,159.752
C09818=1018.335,257.934,367.113,169.281,50.969,159.752
C09819=1018.341,258.183,367.085,169.286,50.963,159.751
C09820=1018.348,258.431,367.057,169.291,50.958,159.751
C09821=1018.354,258.679,367.028,169.295,50.952,159.750
C09822=1018.360,258.928,367.000,169.300,50.946,159.750
C09823=1018.366,259.176,366.973,169.304,50.940,159.749
C09824=1018.372,259.424,366.944,169.309,50.935,159.749
C09825=1018.378,259.673,366.915,169.314,50.929,159.749
C09826=1018.385,259.921,366.888,169.318,50.923,159.748
C09827=1018.391,260.169,366.859,169.323,50.918,159.748
C09828=1018.396,260.418,366.830,169.327,50.912,159.747
C09829=1018.402,260.666,366.801,169.332,50.907,159.747
C09830=1018.408,260.914,366.772,169.337,50.902,159.747
C09831=1018.414,261.163,366.744,169.342,50.896,159.746
C09832=1018.420,261.411,366.715,169.346,50.891,159.746
C09833=1018.426,261.660,366.686,169.351,50.885,159.745
C09834=1018.432,261.907,366.658,169.356,50.879,159.745
C09835=1018.438,262.155,366.628,169.360,50.874,159.744
C09836=1018.444,262.404,366.600,169.365,50.868,159.744
C09837=1018.451,262.652,366.571,169.370,50.863,159.744
C09838=1018.459,262.988,366.532,169.376,50.856,159.743
C09839=1018.467,263.323,366.493,169.383,50.848,159.743
C09840=1018.475,263.658,366.454,169.389,50.841,159.742
C09841=1018.484,263.994,366.415,169.395,50.834,159.742
C09842=1018.490,264.243,366.387,169.400,50.828,159.741
C09843=1018.495,264.491,366.357,169.404,50.823,159.741
C09844=1018.501,264.739,366.328,169.409,50.818,159.741
C09845=1018.508,264.987,366.299,169.413,50.812,159.740
C09846=1018.514,265.236,366.271,169.418,50.807,159.740
C09847=1018.519,265.483,366.242,169.424,50.802,159.740
C09848=1018.525,265.732,366.213,169.428,50.796,159.739
C09849=1018.532,265.980,366.184,169.432,50.791,159.739
C09850=1018.537,266.228,366.154,169.438,50.786,159.738
C09851=1018.543,266.476,366.125,169.442,50.780,159.738
C09852=1018.550,266.724,366.096,169.447,50.775,159.738
C09853=1018.556,266.973,366.067,169.451,50.770,159.737
C09854=1018.561,267.221,366.038,169.457,50.765,159.737
C09855=1018.568,267.469,366.008,169.461,50.759,159.737
C09856=1018.574,267.717,365.979,169.466,50.754,159.736
C09857=1018.580,267.965,365.950,169.470,50.749,159.736
C09858=1018.586,268.214,365.921,169.476,50.744,159.736
C09859=1018.592,268.462,365.892,169.480,50.739,159.735
C09860=1018.598,268.710,365.863,169.485,50.733,159.735
C09861=1018.604,268.958,365.834,169.489,50.728,159.735
C09862=1018.613,269.325,365.790,169.497,50.721,159.734
C09863=1018.623,269.689,365.747,169.503,50.713,159.734
C09864=1018.631,270.055,365.704,169.511,50.706,159.733
C09865=1018.640,270.419,365.660,169.518,50.698,159.733
C09866=1018.646,270.668,365.631,169.523,50.693,159.732
C09867=1018.652,270.916,365.602,169.528,50.688,159.732
C09868=1018.659,271.164,365.572,169.533,50.682,159.732
C09869=1018.665,271.413,365.542,169.537,50.678,159.732
C09870=1018.671,271.661,365.513,169.543,50.673,159.731
C09871=1018.676,271.909,365.483,169.547,50.668,159.731
C09872=1018.683,272.157,365.454,169.552,50.662,159.731
C09873=1018.688,272.405,365.424,169.557,50.657,159.730
C09874=1018.695,272.653,365.395,169.561,50.653,159.730
C09875=1018.701,272.901,365.365,169.567,50.648,159.730
C09876=1018.707,273.149,365.335,169.571,50.643,159.730
C09877=1018.713,273.398,365.305,169.576,50.637,159.729
C09878=1018.719,273.646,365.276,169.581,50.633,159.729
C09879=1018.725,273.894,365.246,169.586,50.628,159.729
C09880=1018.732,274.142,365.216,169.591,50.623,159.729
C09881=1018.737,274.390,365.187,169.596,50.618,159.728
C09882=1018.744,274.639,365.157,169.601,50.613,159.728
C09883=1018.750,274.887,365.127,169.605,50.608,159.728
C09884=1018.756,275.135,365.097,169.611,50.603,159.728
C09885=1018.762,275.383,365.068,169.615,50.599,159.727
C09886=1018.768,275.630,365.038,169.621,50.594,159.727
C09887=1018.774,275.880,365.008,169.625,50.589,159.727
C09888=1018.781,276.127,364.978,169.631,50.584,159.727
C09889=1018.786,276.376,364.948,169.635,50.579,159.726
C09890=1018.793,276.623,364.919,169.641,50.574,159.726
C09891=1018.799,276.872,364.888,169.645,50.570,159.726
C09892=1018.805,277.119,364.858,169.650,50.565,159.726
C09893=1018.812,277.368,364.829,169.655,50.560,159.725
C09894=1018.817,277.596,364.801,169.659,50.555,159.725
C09895=1018.823,277.825,364.772,169.664,50.551,159.725
C09896=1018.828,278.053,364.745,169.668,50.547,159.725
C09897=1018.834,278.282,364.717,169.673,50.543,159.725
C09898=1018.839,278.510,364.689,169.677,50.538,159.724
C09899=1018.845,278.740,364.661,169.682,50.534,159.724
C09900=1018.851,278.968,364.634,169.687,50.529,159.724
C09901=1018.856,279.196,364.605,169.691,50.525,159.724
C09902=1018.862,279.445,364.575,169.696,50.521,159.724
C09903=1018.869,279.693,364.546,169.701,50.516,159.723
C09904=1018.875,279.941,364.515,169.706,50.511,159.723
C09905=1018.881,280.189,364.485,169.712,50.507,159.723
C09906=1018.887,280.437,364.454,169.716,50.502,159.723
C09907=1018.894,280.684,364.425,169.721,50.497,159.723
C09908=1018.900,280.933,364.394,169.726,50.492,159.722
C09909=1018.906,281.181,364.363,169.731,50.488,159.722
C09910=1018.912,281.429,364.333,169.737,50.483,159.722
C09911=1018.919,281.677,364.303,169.741,50.478,159.722
C09912=1018.925,281.925,364.273,169.746,50.474,159.722
C09913=1018.931,282.173,364.242,169.752,50.469,159.722
C09914=1018.937,282.421,364.212,169.756,50.465,159.721
C09915=1018.944,282.669,364.181,169.762,50.460,159.721
C09916=1018.950,282.917,364.151,169.766,50.456,159.721
C09917=1018.956,283.165,364.120,169.771,50.452,159.721
C09918=1018.962,283.413,364.090,169.777,50.447,159.721
C09919=1018.968,283.662,364.059,169.781,50.442,159.720
C09920=1018.975,283.909,364.030,169.787,50.438,159.720
C09921=1018.981,284.158,363.999,169.792,50.433,159.720
C09922=1018.987,284.406,363.968,169.798,50.429,159.720
C09923=1018.994,284.654,363.938,169.802,50.424,159.720
C09924=1019.000,284.902,363.908,169.807,50.420,159.720
C09925=1019.007,285.150,363.877,169.813,50.415,159.720
C09926=1019.013,285.397,363.846,169.817,50.411,159.720
C09927=1019.019,285.646,363.815,169.822,50.407,159.719
C09928=1019.025,285.893,363.784,169.828,50.402,159.719
C09929=1019.032,286.142,363.754,169.833,50.398,159.719
C09930=1019.037,286.390,363.723,169.838,50.393,159.719
C09931=1019.044,286.637,363.692,169.843,50.389,159.719
C09932=1019.050,286.885,363.662,169.848,50.385,159.719
C09933=1019.056,287.134,363.631,169.853,50.380,159.719
C09934=1019.063,287.381,363.600,169.858,50.376,159.719
C09935=1019.069,287.629,363.569,169.864,50.372,159.719
C09936=1019.076,287.877,363.538,169.869,50.368,159.718
C09937=1019.081,288.126,363.507,169.874,50.363,159.718
C09938=1019.087,288.374,363.476,169.880,50.359,159.718
C09939=1019.093,288.621,363.445,169.884,50.355,159.718
C09940=1019.100,288.870,363.414,169.889,50.351,159.718
C09941=1019.106,289.118,363.383,169.895,50.346,159.718
C09942=1019.112,289.365,363.352,169.900,50.342,159.718
C09943=1019.119,289.613,363.321,169.906,50.337,159.718
C09944=1019.126,289.861,363.290,169.910,50.333,159.718
C09945=1019.132,290.109,363.259,169.915,50.329,159.718
C09946=1019.138,290.357,363.228,169.921,50.325,159.718
C09947=1019.145,290.606,363.197,169.926,50.320,159.717
C09948=1019.151,290.853,363.166,169.932,50.316,159.717
C09949=1019.157,291.101,363.134,169.937,50.312,159.717
C09950=1019.163,291.349,363.103,169.941,50.308,159.717
C09951=1019.169,291.597,363.072,169.947,50.304,159.717
C09952=1019.176,291.845,363.041,169.952,50.300,159.717
C09953=1019.182,292.093,363.010,169.957,50.296,159.717
C09954=1019.188,292.328,362.980,169.962,50.292,159.717
C09955=1019.194,292.562,362.950,169.968,50.288,159.717
C09956=1019.200,292.796,362.921,169.973,50.284,159.717
C09957=1019.207,293.031,362.891,169.978,50.280,159.717
C09958=1019.212,293.266,362.861,169.983,50.276,159.717
C09959=1019.218,293.501,362.831,169.988,50.273,159.717
C09960=1019.224,293.736,362.801,169.993,50.269,159.717
C09961=1019.229,293.971,362.771,169.998,50.265,159.717
C09962=1019.236,294.219,362.740,170.003,50.261,159.717
C09963=1019.242,294.467,362.708,170.008,50.257,159.717
C09964=1019.248,294.714,362.676,170.013,50.253,159.717
C09965=1019.254,294.962,362.645,170.019,50.249,159.717
C09966=1019.261,295.210,362.612,170.024,50.246,159.717
C09967=1019.267,295.458,362.581,170.029,50.242,159.717
C09968=1019.273,295.705,362.549,170.035,50.237,159.717
C09969=1019.279,295.953,362.518,170.040,50.233,159.717
C09970=1019.285,296.201,362.486,170.045,50.230,159.717
C09971=1019.292,296.449,362.454,170.051,50.226,159.717
C09972=1019.298,296.697,362.422,170.056,50.222,159.717
C09973=1019.304,296.945,362.389,170.061,50.218,159.717
C09974=1019.311,297.192,362.358,170.067,50.214,159.717
C09975=1019.317,297.440,362.326,170.072,50.211,159.717
C09976=1019.323,297.688,362.295,170.077,50.207,159.717
C09977=1019.330,297.936,362.262,170.083,50.202,159.717
C09978=1019.336,298.184,362.231,170.088,50.199,159.717
C09979=1019.342,298.432,362.199,170.093,50.195,159.717
C09980=1019.348,298.680,362.167,170.100,50.191,159.717
C09981=1019.355,298.928,362.134,170.105,50.187,159.717
C09982=1019.361,299.176,362.102,170.111,50.184,159.717
C09983=1019.368,299.424,362.071,170.116,50.180,159.717
C09984=1019.374,299.671,362.038,170.121,50.176,159.717
C09985=1019.381,299.919,362.007,170.127,50.172,159.717
C09986=1019.387,300.167,361.974,170.132,50.169,159.717
C09987=1019.393,300.414,361.942,170.137,50.165,159.717
C09988=1019.399,300.662,361.911,170.143,50.161,159.717
C09989=1019.406,300.910,361.878,170.148,50.157,159.717
C09990=1019.413,301.158,361.846,170.154,50.154,159.717
C09991=1019.419,301.406,361.814,170.160,50.150,159.718
C09992=1019.426,301.654,361.782,170.165,50.146,159.717
C09993=1019.432,301.901,361.750,170.171,50.143,159.718
C09994=1019.438,302.150,361.718,170.176,50.139,159.718
C09995=1019.445,302.397,361.685,170.181,50.135,159.718
C09996=1019.451,302.645,361.653,170.187,50.132,159.718
//INST
///DATE 2021/06/25 14:50
///ATTR SC,RW,RJ
////FRAME ROBOT
///GROUP1 RB1
NOP
MOVL C00000 V=800.0 PL=0
MOVL C00001 V=800.0 PL=0
MOVL C00002 V=800.0 PL=0
MOVL C00003 V=800.0 PL=0
MOVL C00004 V=800.0 PL=0
MOVL C00005 V=800.0 PL=0
MOVL C00006 V=800.0 PL=0
MOVL C00007 V=800.0 PL=0
MOVL C00008 V=800.0 PL=0
MOVL C00009 V=800.0 PL=0
MOVL C00010 V=800.0 PL=0
MOVL C00011 V=800.0 PL=0
MOVL C00012 V=800.0 PL=0
MOVL C00013 V=800.0 PL=0
MOVL C00014 V=800.0 PL=0
MOVL C00015 V=800.0 PL=0
MOVL C00016 V=800.0 PL=0
MOVL C00017 V=800.0 PL=0
MOVL C00018 V=800.0 PL=0
MOVL C00019 V=800.0 PL=0
MOVL C00020 V=800.0 PL=0
MOVL C00021 V=800.0 PL=0
MOVL C00022 V=800.0 PL=0
MOVL C00023 V=800.0 PL=0
MOVL C00024 V=800.0 PL=0
MOVL C00025 V=800.0 PL=0
MOVL C00026 V=800.0 PL=0
MOVL C00027 V=800.0 PL=0
MOVL C00028 V=800.0 PL=0
MOVL C00029 V=800.0 PL=0
MOVL C00030 V=800.0 PL=0
MOVL C00031 V=800.0 PL=0
MOVL C00032 V=800.0 PL=0
MOVL C00033 V=800.0 PL=0
MOVL C00034 V=800.0 PL=0
MOVL C00035 V=800.0 PL=0
MOVL C00036 V=800.0 PL=0
MOVL C00037 V=800.0 PL=0
MOVL C00038 V=800.0 PL=0
MOVL C00039 V=800.0 PL=0
MOVL C00040 V=800.0 PL=0
MOVL C00041 V=800.0 PL=0
MOVL C00042 V=800.0 PL=0
MOVL C00043 V=800.0 PL=0
MOVL C00044 V=800.0 PL=0
MOVL C00045 V=800.0 PL=0
MOVL C00046 V=800.0 PL=0
MOVL C00047 V=800.0 PL=0
MOVL C00048 V=800.0 PL=0
MOVL C00049 V=800.0 PL=0
MOVL C00050 V=800.0 PL=0
MOVL C00051 V=800.0 PL=0
MOVL C00052 V=800.0 PL=0
MOVL C00053 V=800.0 PL=0
MOVL C00054 V=800.0 PL=0
MOVL C00055 V=800.0 PL=0
MOVL C00056 V=800.0 PL=0
MOVL C00057 V=800.0 PL=0
MOVL C00058 V=800.0 PL=0
MOVL C00059 V=800.0 PL=0
MOVL C00060 V=800.0 PL=0
MOVL C00061 V=800.0 PL=0
MOVL C00062 V=800.0 PL=0
MOVL C00063 V=800.0 PL=0
MOVL C00064 V=800.0 PL=0
MOVL C00065 V=800.0 PL=0
MOVL C00066 V=800.0 PL=0
MOVL C00067 V=800.0 PL=0
MOVL C00068 V=800.0 PL=0
MOVL C00069 V=800.0 PL=0
MOVL C00070 V=800.0 PL=0
MOVL C00071 V=800.0 PL=0
MOVL C00072 V=800.0 PL=0
MOVL C00073 V=800.0 PL=0
MOVL C00074 V=800.0 PL=0
MOVL C00075 V=800.0 PL=0
MOVL C00076 V=800.0 PL=0
MOVL C00077 V=800.0 PL=0
MOVL C00078 V=800.0 PL=0
MOVL C00079 V=800.0 PL=0
MOVL C00080 V=800.0 PL=0
MOVL C00081 V=800.0 PL=0
MOVL C00082 V=800.0 PL=0
MOVL C00083 V=800.0 PL=0
MOVL C00084 V=800.0 PL=0
MOVL C00085 V=800.0 PL=0
MOVL C00086 V=800.0 PL=0
MOVL C00087 V=800.0 PL=0
MOVL C00088 V=800.0 PL=0
MOVL C00089 V=800.0 PL=0
MOVL C00090 V=800.0 PL=0
MOVL C00091 V=800.0 PL=0
MOVL C00092 V=800.0 PL=0
MOVL C00093 V=800.0 PL=0
MOVL C00094 V=800.0 PL=0
MOVL C00095 V=800.0 PL=0
MOVL C00096 V=800.0 PL=0
MOVL C00097 V=800.0 PL=0
MOVL C00098 V=800.0 PL=0
MOVL C00099 V=800.0 PL=0
MOVL C00100 V=800.0 PL=0
MOVL C00101 V=800.0 PL=0
MOVL C00102 V=800.0 PL=0
MOVL C00103 V=800.0 PL=0
MOVL C00104 V=800.0 PL=0
MOVL C00105 V=800.0 PL=0
MOVL C00106 V=800.0 PL=0
MOVL C00107 V=800.0 PL=0
MOVL C00108 V=800.0 PL=0
MOVL C00109 V=800.0 PL=0
MOVL C00110 V=800.0 PL=0
MOVL C00111 V=800.0 PL=0
MOVL C00112 V=800.0 PL=0
MOVL C00113 V=800.0 PL=0
MOVL C00114 V=800.0 PL=0
MOVL C00115 V=800.0 PL=0
MOVL C00116 V=800.0 PL=0
MOVL C00117 V=800.0 PL=0
MOVL C00118 V=800.0 PL=0
MOVL C00119 V=800.0 PL=0
MOVL C00120 V=800.0 PL=0
MOVL C00121 V=800.0 PL=0
MOVL C00122 V=800.0 PL=0
MOVL C00123 V=800.0 PL=0
MOVL C00124 V=800.0 PL=0
MOVL C00125 V=800.0 PL=0
MOVL C00126 V=800.0 PL=0
MOVL C00127 V=800.0 PL=0
MOVL C00128 V=800.0 PL=0
MOVL C00129 V=800.0 PL=0
MOVL C00130 V=800.0 PL=0
MOVL C00131 V=800.0 PL=0
MOVL C00132 V=800.0 PL=0
MOVL C00133 V=800.0 PL=0
MOVL C00134 V=800.0 PL=0
MOVL C00135 V=800.0 PL=0
MOVL C00136 V=800.0 PL=0
MOVL C00137 V=800.0 PL=0
MOVL C00138 V=800.0 PL=0
MOVL C00139 V=800.0 PL=0
MOVL C00140 V=800.0 PL=0
MOVL C00141 V=800.0 PL=0
MOVL C00142 V=800.0 PL=0
MOVL C00143 V=800.0 PL=0
MOVL C00144 V=800.0 PL=0
MOVL C00145 V=800.0 PL=0
MOVL C00146 V=800.0 PL=0
MOVL C00147 V=800.0 PL=0
MOVL C00148 V=800.0 PL=0
MOVL C00149 V=800.0 PL=0
MOVL C00150 V=800.0 PL=0
MOVL C00151 V=800.0 PL=0
MOVL C00152 V=800.0 PL=0
MOVL C00153 V=800.0 PL=0
MOVL C00154 V=800.0 PL=0
MOVL C00155 V=800.0 PL=0
MOVL C00156 V=800.0 PL=0
MOVL C00157 V=800.0 PL=0
MOVL C00158 V=800.0 PL=0
MOVL C00159 V=800.0 PL=0
MOVL C00160 V=800.0 PL=0
MOVL C00161 V=800.0 PL=0
MOVL C00162 V=800.0 PL=0
MOVL C00163 V=800.0 PL=0
MOVL C00164 V=800.0 PL=0
MOVL C00165 V=800.0 PL=0
MOVL C00166 V=800.0 PL=0
MOVL C00167 V=800.0 PL=0
MOVL C00168 V=800.0 PL=0
MOVL C00169 V=800.0 PL=0
MOVL C00170 V=800.0 PL=0
MOVL C00171 V=800.0 PL=0
MOVL C00172 V=800.0 PL=0
MOVL C00173 V=800.0 PL=0
MOVL C00174 V=800.0 PL=0
MOVL C00175 V=800.0 PL=0
MOVL C00176 V=800.0 PL=0
MOVL C00177 V=800.0 PL=0
MOVL C00178 V=800.0 PL=0
MOVL C00179 V=800.0 PL=0
MOVL C00180 V=800.0 PL=0
MOVL C00181 V=800.0 PL=0
MOVL C00182 V=800.0 PL=0
MOVL C00183 V=800.0 PL=0
MOVL C00184 V=800.0 PL=0
MOVL C00185 V=800.0 PL=0
MOVL C00186 V=800.0 PL=0
MOVL C00187 V=800.0 PL=0
MOVL C00188 V=800.0 PL=0
MOVL C00189 V=800.0 PL=0
MOVL C00190 V=800.0 PL=0
MOVL C00191 V=800.0 PL=0
MOVL C00192 V=800.0 PL=0
MOVL C00193 V=800.0 PL=0
MOVL C00194 V=800.0 PL=0
MOVL C00195 V=800.0 PL=0
MOVL C00196 V=800.0 PL=0
MOVL C00197 V=800.0 PL=0
MOVL C00198 V=800.0 PL=0
MOVL C00199 V=800.0 PL=0
MOVL C00200 V=800.0 PL=0
MOVL C00201 V=800.0 PL=0
MOVL C00202 V=800.0 PL=0
MOVL C00203 V=800.0 PL=0
MOVL C00204 V=800.0 PL=0
MOVL C00205 V=800.0 PL=0
MOVL C00206 V=800.0 PL=0
MOVL C00207 V=800.0 PL=0
MOVL C00208 V=800.0 PL=0
MOVL C00209 V=800.0 PL=0
MOVL C00210 V=800.0 PL=0
MOVL C00211 V=800.0 PL=0
MOVL C00212 V=800.0 PL=0
MOVL C00213 V=800.0 PL=0
MOVL C00214 V=800.0 PL=0
MOVL C00215 V=800.0 PL=0
MOVL C00216 V=800.0 PL=0
MOVL C00217 V=800.0 PL=0
MOVL C00218 V=800.0 PL=0
MOVL C00219 V=800.0 PL=0
MOVL C00220 V=800.0 PL=0
MOVL C00221 V=800.0 PL=0
MOVL C00222 V=800.0 PL=0
MOVL C00223 V=800.0 PL=0
MOVL C00224 V=800.0 PL=0
MOVL C00225 V=800.0 PL=0
MOVL C00226 V=800.0 PL=0
MOVL C00227 V=800.0 PL=0
MOVL C00228 V=800.0 PL=0
MOVL C00229 V=800.0 PL=0
MOVL C00230 V=800.0 PL=0
MOVL C00231 V=800.0 PL=0
MOVL C00232 V=800.0 PL=0
MOVL C00233 V=800.0 PL=0
MOVL C00234 V=800.0 PL=0
MOVL C00235 V=800.0 PL=0
MOVL C00236 V=800.0 PL=0
MOVL C00237 V=800.0 PL=0
MOVL C00238 V=800.0 PL=0
MOVL C00239 V=800.0 PL=0
MOVL C00240 V=800.0 PL=0
MOVL C00241 V=800.0 PL=0
MOVL C00242 V=800.0 PL=0
MOVL C00243 V=800.0 PL=0
MOVL C00244 V=800.0 PL=0
MOVL C00245 V=800.0 PL=0
MOVL C00246 V=800.0 PL=0
MOVL C00247 V=800.0 PL=0
MOVL C00248 V=800.0 PL=0
MOVL C00249 V=800.0 PL=0
MOVL C00250 V=800.0 PL=0
MOVL C00251 V=800.0 PL=0
MOVL C00252 V=800.0 PL=0
MOVL C00253 V=800.0 PL=0
MOVL C00254 V=800.0 PL=0
MOVL C00255 V=800.0 PL=0
MOVL C00256 V=800.0 PL=0
MOVL C00257 V=800.0 PL=0
MOVL C00258 V=800.0 PL=0
MOVL C00259 V=800.0 PL=0
MOVL C00260 V=800.0 PL=0
MOVL C00261 V=800.0 PL=0
MOVL C00262 V=800.0 PL=0
MOVL C00263 V=800.0 PL=0
MOVL C00264 V=800.0 PL=0
MOVL C00265 V=800.0 PL=0
MOVL C00266 V=800.0 PL=0
MOVL C00267 V=800.0 PL=0
MOVL C00268 V=800.0 PL=0
MOVL C00269 V=800.0 PL=0
MOVL C00270 V=800.0 PL=0
MOVL C00271 V=800.0 PL=0
MOVL C00272 V=800.0 PL=0
MOVL C00273 V=800.0 PL=0
MOVL C00274 V=800.0 PL=0
MOVL C00275 V=800.0 PL=0
MOVL C00276 V=800.0 PL=0
MOVL C00277 V=800.0 PL=0
MOVL C00278 V=800.0 PL=0
MOVL C00279 V=800.0 PL=0
MOVL C00280 V=800.0 PL=0
MOVL C00281 V=800.0 PL=0
MOVL C00282 V=800.0 PL=0
MOVL C00283 V=800.0 PL=0
MOVL C00284 V=800.0 PL=0
MOVL C00285 V=800.0 PL=0
MOVL C00286 V=800.0 PL=0
MOVL C00287 V=800.0 PL=0
MOVL C00288 V=800.0 PL=0
MOVL C00289 V=800.0 PL=0
MOVL C00290 V=800.0 PL=0
MOVL C00291 V=800.0 PL=0
MOVL C00292 V=800.0 PL=0
MOVL C00293 V=800.0 PL=0
MOVL C00294 V=800.0 PL=0
MOVL C00295 V=800.0 PL=0
MOVL C00296 V=800.0 PL=0
MOVL C00297 V=800.0 PL=0
MOVL C00298 V=800.0 PL=0
MOVL C00299 V=800.0 PL=0
MOVL C00300 V=800.0 PL=0
MOVL C00301 V=800.0 PL=0
MOVL C00302 V=800.0 PL=0
MOVL C00303 V=800.0 PL=0
MOVL C00304 V=800.0 PL=0
MOVL C00305 V=800.0 PL=0
MOVL C00306 V=800.0 PL=0
MOVL C00307 V=800.0 PL=0
MOVL C00308 V=800.0 PL=0
MOVL C00309 V=800.0 PL=0
MOVL C00310 V=800.0 PL=0
MOVL C00311 V=800.0 PL=0
MOVL C00312 V=800.0 PL=0
MOVL C00313 V=800.0 PL=0
MOVL C00314 V=800.0 PL=0
MOVL C00315 V=800.0 PL=0
MOVL C00316 V=800.0 PL=0
MOVL C00317 V=800.0 PL=0
MOVL C00318 V=800.0 PL=0
MOVL C00319 V=800.0 PL=0
MOVL C00320 V=800.0 PL=0
MOVL C00321 V=800.0 PL=0
MOVL C00322 V=800.0 PL=0
MOVL C00323 V=800.0 PL=0
MOVL C00324 V=800.0 PL=0
MOVL C00325 V=800.0 PL=0
MOVL C00326 V=800.0 PL=0
MOVL C00327 V=800.0 PL=0
MOVL C00328 V=800.0 PL=0
MOVL C00329 V=800.0 PL=0
MOVL C00330 V=800.0 PL=0
MOVL C00331 V=800.0 PL=0
MOVL C00332 V=800.0 PL=0
MOVL C00333 V=800.0 PL=0
MOVL C00334 V=800.0 PL=0
MOVL C00335 V=800.0 PL=0
MOVL C00336 V=800.0 PL=0
MOVL C00337 V=800.0 PL=0
MOVL C00338 V=800.0 PL=0
MOVL C00339 V=800.0 PL=0
MOVL C00340 V=800.0 PL=0
MOVL C00341 V=800.0 PL=0
MOVL C00342 V=800.0 PL=0
MOVL C00343 V=800.0 PL=0
MOVL C00344 V=800.0 PL=0
MOVL C00345 V=800.0 PL=0
MOVL C00346 V=800.0 PL=0
MOVL C00347 V=800.0 PL=0
MOVL C00348 V=800.0 PL=0
MOVL C00349 V=800.0 PL=0
MOVL C00350 V=800.0 PL=0
MOVL C00351 V=800.0 PL=0
MOVL C00352 V=800.0 PL=0
MOVL C00353 V=800.0 PL=0
MOVL C00354 V=800.0 PL=0
MOVL C00355 V=800.0 PL=0
MOVL C00356 V=800.0 PL=0
MOVL C00357 V=800.0 PL=0
MOVL C00358 V=800.0 PL=0
MOVL C00359 V=800.0 PL=0
MOVL C00360 V=800.0 PL=0
MOVL C00361 V=800.0 PL=0
MOVL C00362 V=800.0 PL=0
MOVL C00363 V=800.0 PL=0
MOVL C00364 V=800.0 PL=0
MOVL C00365 V=800.0 PL=0
MOVL C00366 V=800.0 PL=0
MOVL C00367 V=800.0 PL=0
MOVL C00368 V=800.0 PL=0
MOVL C00369 V=800.0 PL=0
MOVL C00370 V=800.0 PL=0
MOVL C00371 V=800.0 PL=0
MOVL C00372 V=800.0 PL=0
MOVL C00373 V=800.0 PL=0
MOVL C00374 V=800.0 PL=0
MOVL C00375 V=800.0 PL=0
MOVL C00376 V=800.0 PL=0
MOVL C00377 V=800.0 PL=0
MOVL C00378 V=800.0 PL=0
MOVL C00379 V=800.0 PL=0
MOVL C00380 V=800.0 PL=0
MOVL C00381 V=800.0 PL=0
MOVL C00382 V=800.0 PL=0
MOVL C00383 V=800.0 PL=0
MOVL C00384 V=800.0 PL=0
MOVL C00385 V=800.0 PL=0
MOVL C00386 V=800.0 PL=0
MOVL C00387 V=800.0 PL=0
MOVL C00388 V=800.0 PL=0
MOVL C00389 V=800.0 PL=0
MOVL C00390 V=800.0 PL=0
MOVL C00391 V=800.0 PL=0
MOVL C00392 V=800.0 PL=0
MOVL C00393 V=800.0 PL=0
MOVL C00394 V=800.0 PL=0
MOVL C00395 V=800.0 PL=0
MOVL C00396 V=800.0 PL=0
MOVL C00397 V=800.0 PL=0
MOVL C00398 V=800.0 PL=0
MOVL C00399 V=800.0 PL=0
MOVL C00400 V=800.0 PL=0
MOVL C00401 V=800.0 PL=0
MOVL C00402 V=800.0 PL=0
MOVL C00403 V=800.0 PL=0
MOVL C00404 V=800.0 PL=0
MOVL C00405 V=800.0 PL=0
MOVL C00406 V=800.0 PL=0
MOVL C00407 V=800.0 PL=0
MOVL C00408 V=800.0 PL=0
MOVL C00409 V=800.0 PL=0
MOVL C00410 V=800.0 PL=0
MOVL C00411 V=800.0 PL=0
MOVL C00412 V=800.0 PL=0
MOVL C00413 V=800.0 PL=0
MOVL C00414 V=800.0 PL=0
MOVL C00415 V=800.0 PL=0
MOVL C00416 V=800.0 PL=0
MOVL C00417 V=800.0 PL=0
MOVL C00418 V=800.0 PL=0
MOVL C00419 V=800.0 PL=0
MOVL C00420 V=800.0 PL=0
MOVL C00421 V=800.0 PL=0
MOVL C00422 V=800.0 PL=0
MOVL C00423 V=800.0 PL=0
MOVL C00424 V=800.0 PL=0
MOVL C00425 V=800.0 PL=0
MOVL C00426 V=800.0 PL=0
MOVL C00427 V=800.0 PL=0
MOVL C00428 V=800.0 PL=0
MOVL C00429 V=800.0 PL=0
MOVL C00430 V=800.0 PL=0
MOVL C00431 V=800.0 PL=0
MOVL C00432 V=800.0 PL=0
MOVL C00433 V=800.0 PL=0
MOVL C00434 V=800.0 PL=0
MOVL C00435 V=800.0 PL=0
MOVL C00436 V=800.0 PL=0
MOVL C00437 V=800.0 PL=0
MOVL C00438 V=800.0 PL=0
MOVL C00439 V=800.0 PL=0
MOVL C00440 V=800.0 PL=0
MOVL C00441 V=800.0 PL=0
MOVL C00442 V=800.0 PL=0
MOVL C00443 V=800.0 PL=0
MOVL C00444 V=800.0 PL=0
MOVL C00445 V=800.0 PL=0
MOVL C00446 V=800.0 PL=0
MOVL C00447 V=800.0 PL=0
MOVL C00448 V=800.0 PL=0
MOVL C00449 V=800.0 PL=0
MOVL C00450 V=800.0 PL=0
MOVL C00451 V=800.0 PL=0
MOVL C00452 V=800.0 PL=0
MOVL C00453 V=800.0 PL=0
MOVL C00454 V=800.0 PL=0
MOVL C00455 V=800.0 PL=0
MOVL C00456 V=800.0 PL=0
MOVL C00457 V=800.0 PL=0
MOVL C00458 V=800.0 PL=0
MOVL C00459 V=800.0 PL=0
MOVL C00460 V=800.0 PL=0
MOVL C00461 V=800.0 PL=0
MOVL C00462 V=800.0 PL=0
MOVL C00463 V=800.0 PL=0
MOVL C00464 V=800.0 PL=0
MOVL C00465 V=800.0 PL=0
MOVL C00466 V=800.0 PL=0
MOVL C00467 V=800.0 PL=0
MOVL C00468 V=800.0 PL=0
MOVL C00469 V=800.0 PL=0
MOVL C00470 V=800.0 PL=0
MOVL C00471 V=800.0 PL=0
MOVL C00472 V=800.0 PL=0
MOVL C00473 V=800.0 PL=0
MOVL C00474 V=800.0 PL=0
MOVL C00475 V=800.0 PL=0
MOVL C00476 V=800.0 PL=0
MOVL C00477 V=800.0 PL=0
MOVL C00478 V=800.0 PL=0
MOVL C00479 V=800.0 PL=0
MOVL C00480 V=800.0 PL=0
MOVL C00481 V=800.0 PL=0
MOVL C00482 V=800.0 PL=0
MOVL C00483 V=800.0 PL=0
MOVL C00484 V=800.0 PL=0
MOVL C00485 V=800.0 PL=0
MOVL C00486 V=800.0 PL=0
MOVL C00487 V=800.0 PL=0
MOVL C00488 V=800.0 PL=0
MOVL C00489 V=800.0 PL=0
MOVL C00490 V=800.0 PL=0
MOVL C00491 V=800.0 PL=0
MOVL C00492 V=800.0 PL=0
MOVL C00493 V=800.0 PL=0
MOVL C00494 V=800.0 PL=0
MOVL C00495 V=800.0 PL=0
MOVL C00496 V=800.0 PL=0
MOVL C00497 V=800.0 PL=0
MOVL C00498 V=800.0 PL=0
MOVL C00499 V=800.0 PL=0
MOVL C00500 V=800.0 PL=0
MOVL C00501 V=800.0 PL=0
MOVL C00502 V=800.0 PL=0
MOVL C00503 V=800.0 PL=0
MOVL C00504 V=800.0 PL=0
MOVL C00505 V=800.0 PL=0
MOVL C00506 V=800.0 PL=0
MOVL C00507 V=800.0 PL=0
MOVL C00508 V=800.0 PL=0
MOVL C00509 V=800.0 PL=0
MOVL C00510 V=800.0 PL=0
MOVL C00511 V=800.0 PL=0
MOVL C00512 V=800.0 PL=0
MOVL C00513 V=800.0 PL=0
MOVL C00514 V=800.0 PL=0
MOVL C00515 V=800.0 PL=0
MOVL C00516 V=800.0 PL=0
MOVL C00517 V=800.0 PL=0
MOVL C00518 V=800.0 PL=0
MOVL C00519 V=800.0 PL=0
MOVL C00520 V=800.0 PL=0
MOVL C00521 V=800.0 PL=0
MOVL C00522 V=800.0 PL=0
MOVL C00523 V=800.0 PL=0
MOVL C00524 V=800.0 PL=0
MOVL C00525 V=800.0 PL=0
MOVL C00526 V=800.0 PL=0
MOVL C00527 V=800.0 PL=0
MOVL C00528 V=800.0 PL=0
MOVL C00529 V=800.0 PL=0
MOVL C00530 V=800.0 PL=0
MOVL C00531 V=800.0 PL=0
MOVL C00532 V=800.0 PL=0
MOVL C00533 V=800.0 PL=0
MOVL C00534 V=800.0 PL=0
MOVL C00535 V=800.0 PL=0
MOVL C00536 V=800.0 PL=0
MOVL C00537 V=800.0 PL=0
MOVL C00538 V=800.0 PL=0
MOVL C00539 V=800.0 PL=0
MOVL C00540 V=800.0 PL=0
MOVL C00541 V=800.0 PL=0
MOVL C00542 V=800.0 PL=0
MOVL C00543 V=800.0 PL=0
MOVL C00544 V=800.0 PL=0
MOVL C00545 V=800.0 PL=0
MOVL C00546 V=800.0 PL=0
MOVL C00547 V=800.0 PL=0
MOVL C00548 V=800.0 PL=0
MOVL C00549 V=800.0 PL=0
MOVL C00550 V=800.0 PL=0
MOVL C00551 V=800.0 PL=0
MOVL C00552 V=800.0 PL=0
MOVL C00553 V=800.0 PL=0
MOVL C00554 V=800.0 PL=0
MOVL C00555 V=800.0 PL=0
MOVL C00556 V=800.0 PL=0
MOVL C00557 V=800.0 PL=0
MOVL C00558 V=800.0 PL=0
MOVL C00559 V=800.0 PL=0
MOVL C00560 V=800.0 PL=0
MOVL C00561 V=800.0 PL=0
MOVL C00562 V=800.0 PL=0
MOVL C00563 V=800.0 PL=0
MOVL C00564 V=800.0 PL=0
MOVL C00565 V=800.0 PL=0
MOVL C00566 V=800.0 PL=0
MOVL C00567 V=800.0 PL=0
MOVL C00568 V=800.0 PL=0
MOVL C00569 V=800.0 PL=0
MOVL C00570 V=800.0 PL=0
MOVL C00571 V=800.0 PL=0
MOVL C00572 V=800.0 PL=0
MOVL C00573 V=800.0 PL=0
MOVL C00574 V=800.0 PL=0
MOVL C00575 V=800.0 PL=0
MOVL C00576 V=800.0 PL=0
MOVL C00577 V=800.0 PL=0
MOVL C00578 V=800.0 PL=0
MOVL C00579 V=800.0 PL=0
MOVL C00580 V=800.0 PL=0
MOVL C00581 V=800.0 PL=0
MOVL C00582 V=800.0 PL=0
MOVL C00583 V=800.0 PL=0
MOVL C00584 V=800.0 PL=0
MOVL C00585 V=800.0 PL=0
MOVL C00586 V=800.0 PL=0
MOVL C00587 V=800.0 PL=0
MOVL C00588 V=800.0 PL=0
MOVL C00589 V=800.0 PL=0
MOVL C00590 V=800.0 PL=0
MOVL C00591 V=800.0 PL=0
MOVL C00592 V=800.0 PL=0
MOVL C00593 V=800.0 PL=0
MOVL C00594 V=800.0 PL=0
MOVL C00595 V=800.0 PL=0
MOVL C00596 V=800.0 PL=0
MOVL C00597 V=800.0 PL=0
MOVL C00598 V=800.0 PL=0
MOVL C00599 V=800.0 PL=0
MOVL C00600 V=800.0 PL=0
MOVL C00601 V=800.0 PL=0
MOVL C00602 V=800.0 PL=0
MOVL C00603 V=800.0 PL=0
MOVL C00604 V=800.0 PL=0
MOVL C00605 V=800.0 PL=0
MOVL C00606 V=800.0 PL=0
MOVL C00607 V=800.0 PL=0
MOVL C00608 V=800.0 PL=0
MOVL C00609 V=800.0 PL=0
MOVL C00610 V=800.0 PL=0
MOVL C00611 V=800.0 PL=0
MOVL C00612 V=800.0 PL=0
MOVL C00613 V=800.0 PL=0
MOVL C00614 V=800.0 PL=0
MOVL C00615 V=800.0 PL=0
MOVL C00616 V=800.0 PL=0
MOVL C00617 V=800.0 PL=0
MOVL C00618 V=800.0 PL=0
MOVL C00619 V=800.0 PL=0
MOVL C00620 V=800.0 PL=0
MOVL C00621 V=800.0 PL=0
MOVL C00622 V=800.0 PL=0
MOVL C00623 V=800.0 PL=0
MOVL C00624 V=800.0 PL=0
MOVL C00625 V=800.0 PL=0
MOVL C00626 V=800.0 PL=0
MOVL C00627 V=800.0 PL=0
MOVL C00628 V=800.0 PL=0
MOVL C00629 V=800.0 PL=0
MOVL C00630 V=800.0 PL=0
MOVL C00631 V=800.0 PL=0
MOVL C00632 V=800.0 PL=0
MOVL C00633 V=800.0 PL=0
MOVL C00634 V=800.0 PL=0
MOVL C00635 V=800.0 PL=0
MOVL C00636 V=800.0 PL=0
MOVL C00637 V=800.0 PL=0
MOVL C00638 V=800.0 PL=0
MOVL C00639 V=800.0 PL=0
MOVL C00640 V=800.0 PL=0
MOVL C00641 V=800.0 PL=0
MOVL C00642 V=800.0 PL=0
MOVL C00643 V=800.0 PL=0
MOVL C00644 V=800.0 PL=0
MOVL C00645 V=800.0 PL=0
MOVL C00646 V=800.0 PL=0
MOVL C00647 V=800.0 PL=0
MOVL C00648 V=800.0 PL=0
MOVL C00649 V=800.0 PL=0
MOVL C00650 V=800.0 PL=0
MOVL C00651 V=800.0 PL=0
MOVL C00652 V=800.0 PL=0
MOVL C00653 V=800.0 PL=0
MOVL C00654 V=800.0 PL=0
MOVL C00655 V=800.0 PL=0
MOVL C00656 V=800.0 PL=0
MOVL C00657 V=800.0 PL=0
MOVL C00658 V=800.0 PL=0
MOVL C00659 V=800.0 PL=0
MOVL C00660 V=800.0 PL=0
MOVL C00661 V=800.0 PL=0
MOVL C00662 V=800.0 PL=0
MOVL C00663 V=800.0 PL=0
MOVL C00664 V=800.0 PL=0
MOVL C00665 V=800.0 PL=0
MOVL C00666 V=800.0 PL=0
MOVL C00667 V=800.0 PL=0
MOVL C00668 V=800.0 PL=0
MOVL C00669 V=800.0 PL=0
MOVL C00670 V=800.0 PL=0
MOVL C00671 V=800.0 PL=0
MOVL C00672 V=800.0 PL=0
MOVL C00673 V=800.0 PL=0
MOVL C00674 V=800.0 PL=0
MOVL C00675 V=800.0 PL=0
MOVL C00676 V=800.0 PL=0
MOVL C00677 V=800.0 PL=0
MOVL C00678 V=800.0 PL=0
MOVL C00679 V=800.0 PL=0
MOVL C00680 V=800.0 PL=0
MOVL C00681 V=800.0 PL=0
MOVL C00682 V=800.0 PL=0
MOVL C00683 V=800.0 PL=0
MOVL C00684 V=800.0 PL=0
MOVL C00685 V=800.0 PL=0
MOVL C00686 V=800.0 PL=0
MOVL C00687 V=800.0 PL=0
MOVL C00688 V=800.0 PL=0
MOVL C00689 V=800.0 PL=0
MOVL C00690 V=800.0 PL=0
MOVL C00691 V=800.0 PL=0
MOVL C00692 V=800.0 PL=0
MOVL C00693 V=800.0 PL=0
MOVL C00694 V=800.0 PL=0
MOVL C00695 V=800.0 PL=0
MOVL C00696 V=800.0 PL=0
MOVL C00697 V=800.0 PL=0
MOVL C00698 V=800.0 PL=0
MOVL C00699 V=800.0 PL=0
MOVL C00700 V=800.0 PL=0
MOVL C00701 V=800.0 PL=0
MOVL C00702 V=800.0 PL=0
MOVL C00703 V=800.0 PL=0
MOVL C00704 V=800.0 PL=0
MOVL C00705 V=800.0 PL=0
MOVL C00706 V=800.0 PL=0
MOVL C00707 V=800.0 PL=0
MOVL C00708 V=800.0 PL=0
MOVL C00709 V=800.0 PL=0
MOVL C00710 V=800.0 PL=0
MOVL C00711 V=800.0 PL=0
MOVL C00712 V=800.0 PL=0
MOVL C00713 V=800.0 PL=0
MOVL C00714 V=800.0 PL=0
MOVL C00715 V=800.0 PL=0
MOVL C00716 V=800.0 PL=0
MOVL C00717 V=800.0 PL=0
MOVL C00718 V=800.0 PL=0
MOVL C00719 V=800.0 PL=0
MOVL C00720 V=800.0 PL=0
MOVL C00721 V=800.0 PL=0
MOVL C00722 V=800.0 PL=0
MOVL C00723 V=800.0 PL=0
MOVL C00724 V=800.0 PL=0
MOVL C00725 V=800.0 PL=0
MOVL C00726 V=800.0 PL=0
MOVL C00727 V=800.0 PL=0
MOVL C00728 V=800.0 PL=0
MOVL C00729 V=800.0 PL=0
MOVL C00730 V=800.0 PL=0
MOVL C00731 V=800.0 PL=0
MOVL C00732 V=800.0 PL=0
MOVL C00733 V=800.0 PL=0
MOVL C00734 V=800.0 PL=0
MOVL C00735 V=800.0 PL=0
MOVL C00736 V=800.0 PL=0
MOVL C00737 V=800.0 PL=0
MOVL C00738 V=800.0 PL=0
MOVL C00739 V=800.0 PL=0
MOVL C00740 V=800.0 PL=0
MOVL C00741 V=800.0 PL=0
MOVL C00742 V=800.0 PL=0
MOVL C00743 V=800.0 PL=0
MOVL C00744 V=800.0 PL=0
MOVL C00745 V=800.0 PL=0
MOVL C00746 V=800.0 PL=0
MOVL C00747 V=800.0 PL=0
MOVL C00748 V=800.0 PL=0
MOVL C00749 V=800.0 PL=0
MOVL C00750 V=800.0 PL=0
MOVL C00751 V=800.0 PL=0
MOVL C00752 V=800.0 PL=0
MOVL C00753 V=800.0 PL=0
MOVL C00754 V=800.0 PL=0
MOVL C00755 V=800.0 PL=0
MOVL C00756 V=800.0 PL=0
MOVL C00757 V=800.0 PL=0
MOVL C00758 V=800.0 PL=0
MOVL C00759 V=800.0 PL=0
MOVL C00760 V=800.0 PL=0
MOVL C00761 V=800.0 PL=0
MOVL C00762 V=800.0 PL=0
MOVL C00763 V=800.0 PL=0
MOVL C00764 V=800.0 PL=0
MOVL C00765 V=800.0 PL=0
MOVL C00766 V=800.0 PL=0
MOVL C00767 V=800.0 PL=0
MOVL C00768 V=800.0 PL=0
MOVL C00769 V=800.0 PL=0
MOVL C00770 V=800.0 PL=0
MOVL C00771 V=800.0 PL=0
MOVL C00772 V=800.0 PL=0
MOVL C00773 V=800.0 PL=0
MOVL C00774 V=800.0 PL=0
MOVL C00775 V=800.0 PL=0
MOVL C00776 V=800.0 PL=0
MOVL C00777 V=800.0 PL=0
MOVL C00778 V=800.0 PL=0
MOVL C00779 V=800.0 PL=0
MOVL C00780 V=800.0 PL=0
MOVL C00781 V=800.0 PL=0
MOVL C00782 V=800.0 PL=0
MOVL C00783 V=800.0 PL=0
MOVL C00784 V=800.0 PL=0
MOVL C00785 V=800.0 PL=0
MOVL C00786 V=800.0 PL=0
MOVL C00787 V=800.0 PL=0
MOVL C00788 V=800.0 PL=0
MOVL C00789 V=800.0 PL=0
MOVL C00790 V=800.0 PL=0
MOVL C00791 V=800.0 PL=0
MOVL C00792 V=800.0 PL=0
MOVL C00793 V=800.0 PL=0
MOVL C00794 V=800.0 PL=0
MOVL C00795 V=800.0 PL=0
MOVL C00796 V=800.0 PL=0
MOVL C00797 V=800.0 PL=0
MOVL C00798 V=800.0 PL=0
MOVL C00799 V=800.0 PL=0
MOVL C00800 V=800.0 PL=0
MOVL C00801 V=800.0 PL=0
MOVL C00802 V=800.0 PL=0
MOVL C00803 V=800.0 PL=0
MOVL C00804 V=800.0 PL=0
MOVL C00805 V=800.0 PL=0
MOVL C00806 V=800.0 PL=0
MOVL C00807 V=800.0 PL=0
MOVL C00808 V=800.0 PL=0
MOVL C00809 V=800.0 PL=0
MOVL C00810 V=800.0 PL=0
MOVL C00811 V=800.0 PL=0
MOVL C00812 V=800.0 PL=0
MOVL C00813 V=800.0 PL=0
MOVL C00814 V=800.0 PL=0
MOVL C00815 V=800.0 PL=0
MOVL C00816 V=800.0 PL=0
MOVL C00817 V=800.0 PL=0
MOVL C00818 V=800.0 PL=0
MOVL C00819 V=800.0 PL=0
MOVL C00820 V=800.0 PL=0
MOVL C00821 V=800.0 PL=0
MOVL C00822 V=800.0 PL=0
MOVL C00823 V=800.0 PL=0
MOVL C00824 V=800.0 PL=0
MOVL C00825 V=800.0 PL=0
MOVL C00826 V=800.0 PL=0
MOVL C00827 V=800.0 PL=0
MOVL C00828 V=800.0 PL=0
MOVL C00829 V=800.0 PL=0
MOVL C00830 V=800.0 PL=0
MOVL C00831 V=800.0 PL=0
MOVL C00832 V=800.0 PL=0
MOVL C00833 V=800.0 PL=0
MOVL C00834 V=800.0 PL=0
MOVL C00835 V=800.0 PL=0
MOVL C00836 V=800.0 PL=0
MOVL C00837 V=800.0 PL=0
MOVL C00838 V=800.0 PL=0
MOVL C00839 V=800.0 PL=0
MOVL C00840 V=800.0 PL=0
MOVL C00841 V=800.0 PL=0
MOVL C00842 V=800.0 PL=0
MOVL C00843 V=800.0 PL=0
MOVL C00844 V=800.0 PL=0
MOVL C00845 V=800.0 PL=0
MOVL C00846 V=800.0 PL=0
MOVL C00847 V=800.0 PL=0
MOVL C00848 V=800.0 PL=0
MOVL C00849 V=800.0 PL=0
MOVL C00850 V=800.0 PL=0
MOVL C00851 V=800.0 PL=0
MOVL C00852 V=800.0 PL=0
MOVL C00853 V=800.0 PL=0
MOVL C00854 V=800.0 PL=0
MOVL C00855 V=800.0 PL=0
MOVL C00856 V=800.0 PL=0
MOVL C00857 V=800.0 PL=0
MOVL C00858 V=800.0 PL=0
MOVL C00859 V=800.0 PL=0
MOVL C00860 V=800.0 PL=0
MOVL C00861 V=800.0 PL=0
MOVL C00862 V=800.0 PL=0
MOVL C00863 V=800.0 PL=0
MOVL C00864 V=800.0 PL=0
MOVL C00865 V=800.0 PL=0
MOVL C00866 V=800.0 PL=0
MOVL C00867 V=800.0 PL=0
MOVL C00868 V=800.0 PL=0
MOVL C00869 V=800.0 PL=0
MOVL C00870 V=800.0 PL=0
MOVL C00871 V=800.0 PL=0
MOVL C00872 V=800.0 PL=0
MOVL C00873 V=800.0 PL=0
MOVL C00874 V=800.0 PL=0
MOVL C00875 V=800.0 PL=0
MOVL C00876 V=800.0 PL=0
MOVL C00877 V=800.0 PL=0
MOVL C00878 V=800.0 PL=0
MOVL C00879 V=800.0 PL=0
MOVL C00880 V=800.0 PL=0
MOVL C00881 V=800.0 PL=0
MOVL C00882 V=800.0 PL=0
MOVL C00883 V=800.0 PL=0
MOVL C00884 V=800.0 PL=0
MOVL C00885 V=800.0 PL=0
MOVL C00886 V=800.0 PL=0
MOVL C00887 V=800.0 PL=0
MOVL C00888 V=800.0 PL=0
MOVL C00889 V=800.0 PL=0
MOVL C00890 V=800.0 PL=0
MOVL C00891 V=800.0 PL=0
MOVL C00892 V=800.0 PL=0
MOVL C00893 V=800.0 PL=0
MOVL C00894 V=800.0 PL=0
MOVL C00895 V=800.0 PL=0
MOVL C00896 V=800.0 PL=0
MOVL C00897 V=800.0 PL=0
MOVL C00898 V=800.0 PL=0
MOVL C00899 V=800.0 PL=0
MOVL C00900 V=800.0 PL=0
MOVL C00901 V=800.0 PL=0
MOVL C00902 V=800.0 PL=0
MOVL C00903 V=800.0 PL=0
MOVL C00904 V=800.0 PL=0
MOVL C00905 V=800.0 PL=0
MOVL C00906 V=800.0 PL=0
MOVL C00907 V=800.0 PL=0
MOVL C00908 V=800.0 PL=0
MOVL C00909 V=800.0 PL=0
MOVL C00910 V=800.0 PL=0
MOVL C00911 V=800.0 PL=0
MOVL C00912 V=800.0 PL=0
MOVL C00913 V=800.0 PL=0
MOVL C00914 V=800.0 PL=0
MOVL C00915 V=800.0 PL=0
MOVL C00916 V=800.0 PL=0
MOVL C00917 V=800.0 PL=0
MOVL C00918 V=800.0 PL=0
MOVL C00919 V=800.0 PL=0
MOVL C00920 V=800.0 PL=0
MOVL C00921 V=800.0 PL=0
MOVL C00922 V=800.0 PL=0
MOVL C00923 V=800.0 PL=0
MOVL C00924 V=800.0 PL=0
MOVL C00925 V=800.0 PL=0
MOVL C00926 V=800.0 PL=0
MOVL C00927 V=800.0 PL=0
MOVL C00928 V=800.0 PL=0
MOVL C00929 V=800.0 PL=0
MOVL C00930 V=800.0 PL=0
MOVL C00931 V=800.0 PL=0
MOVL C00932 V=800.0 PL=0
MOVL C00933 V=800.0 PL=0
MOVL C00934 V=800.0 PL=0
MOVL C00935 V=800.0 PL=0
MOVL C00936 V=800.0 PL=0
MOVL C00937 V=800.0 PL=0
MOVL C00938 V=800.0 PL=0
MOVL C00939 V=800.0 PL=0
MOVL C00940 V=800.0 PL=0
MOVL C00941 V=800.0 PL=0
MOVL C00942 V=800.0 PL=0
MOVL C00943 V=800.0 PL=0
MOVL C00944 V=800.0 PL=0
MOVL C00945 V=800.0 PL=0
MOVL C00946 V=800.0 PL=0
MOVL C00947 V=800.0 PL=0
MOVL C00948 V=800.0 PL=0
MOVL C00949 V=800.0 PL=0
MOVL C00950 V=800.0 PL=0
MOVL C00951 V=800.0 PL=0
MOVL C00952 V=800.0 PL=0
MOVL C00953 V=800.0 PL=0
MOVL C00954 V=800.0 PL=0
MOVL C00955 V=800.0 PL=0
MOVL C00956 V=800.0 PL=0
MOVL C00957 V=800.0 PL=0
MOVL C00958 V=800.0 PL=0
MOVL C00959 V=800.0 PL=0
MOVL C00960 V=800.0 PL=0
MOVL C00961 V=800.0 PL=0
MOVL C00962 V=800.0 PL=0
MOVL C00963 V=800.0 PL=0
MOVL C00964 V=800.0 PL=0
MOVL C00965 V=800.0 PL=0
MOVL C00966 V=800.0 PL=0
MOVL C00967 V=800.0 PL=0
MOVL C00968 V=800.0 PL=0
MOVL C00969 V=800.0 PL=0
MOVL C00970 V=800.0 PL=0
MOVL C00971 V=800.0 PL=0
MOVL C00972 V=800.0 PL=0
MOVL C00973 V=800.0 PL=0
MOVL C00974 V=800.0 PL=0
MOVL C00975 V=800.0 PL=0
MOVL C00976 V=800.0 PL=0
MOVL C00977 V=800.0 PL=0
MOVL C00978 V=800.0 PL=0
MOVL C00979 V=800.0 PL=0
MOVL C00980 V=800.0 PL=0
MOVL C00981 V=800.0 PL=0
MOVL C00982 V=800.0 PL=0
MOVL C00983 V=800.0 PL=0
MOVL C00984 V=800.0 PL=0
MOVL C00985 V=800.0 PL=0
MOVL C00986 V=800.0 PL=0
MOVL C00987 V=800.0 PL=0
MOVL C00988 V=800.0 PL=0
MOVL C00989 V=800.0 PL=0
MOVL C00990 V=800.0 PL=0
MOVL C00991 V=800.0 PL=0
MOVL C00992 V=800.0 PL=0
MOVL C00993 V=800.0 PL=0
MOVL C00994 V=800.0 PL=0
MOVL C00995 V=800.0 PL=0
MOVL C00996 V=800.0 PL=0
MOVL C00997 V=800.0 PL=0
MOVL C00998 V=800.0 PL=0
MOVL C00999 V=800.0 PL=0
MOVL C01000 V=800.0 PL=0
MOVL C01001 V=800.0 PL=0
MOVL C01002 V=800.0 PL=0
MOVL C01003 V=800.0 PL=0
MOVL C01004 V=800.0 PL=0
MOVL C01005 V=800.0 PL=0
MOVL C01006 V=800.0 PL=0
MOVL C01007 V=800.0 PL=0
MOVL C01008 V=800.0 PL=0
MOVL C01009 V=800.0 PL=0
MOVL C01010 V=800.0 PL=0
MOVL C01011 V=800.0 PL=0
MOVL C01012 V=800.0 PL=0
MOVL C01013 V=800.0 PL=0
MOVL C01014 V=800.0 PL=0
MOVL C01015 V=800.0 PL=0
MOVL C01016 V=800.0 PL=0
MOVL C01017 V=800.0 PL=0
MOVL C01018 V=800.0 PL=0
MOVL C01019 V=800.0 PL=0
MOVL C01020 V=800.0 PL=0
MOVL C01021 V=800.0 PL=0
MOVL C01022 V=800.0 PL=0
MOVL C01023 V=800.0 PL=0
MOVL C01024 V=800.0 PL=0
MOVL C01025 V=800.0 PL=0
MOVL C01026 V=800.0 PL=0
MOVL C01027 V=800.0 PL=0
MOVL C01028 V=800.0 PL=0
MOVL C01029 V=800.0 PL=0
MOVL C01030 V=800.0 PL=0
MOVL C01031 V=800.0 PL=0
MOVL C01032 V=800.0 PL=0
MOVL C01033 V=800.0 PL=0
MOVL C01034 V=800.0 PL=0
MOVL C01035 V=800.0 PL=0
MOVL C01036 V=800.0 PL=0
MOVL C01037 V=800.0 PL=0
MOVL C01038 V=800.0 PL=0
MOVL C01039 V=800.0 PL=0
MOVL C01040 V=800.0 PL=0
MOVL C01041 V=800.0 PL=0
MOVL C01042 V=800.0 PL=0
MOVL C01043 V=800.0 PL=0
MOVL C01044 V=800.0 PL=0
MOVL C01045 V=800.0 PL=0
MOVL C01046 V=800.0 PL=0
MOVL C01047 V=800.0 PL=0
MOVL C01048 V=800.0 PL=0
MOVL C01049 V=800.0 PL=0
MOVL C01050 V=800.0 PL=0
MOVL C01051 V=800.0 PL=0
MOVL C01052 V=800.0 PL=0
MOVL C01053 V=800.0 PL=0
MOVL C01054 V=800.0 PL=0
MOVL C01055 V=800.0 PL=0
MOVL C01056 V=800.0 PL=0
MOVL C01057 V=800.0 PL=0
MOVL C01058 V=800.0 PL=0
MOVL C01059 V=800.0 PL=0
MOVL C01060 V=800.0 PL=0
MOVL C01061 V=800.0 PL=0
MOVL C01062 V=800.0 PL=0
MOVL C01063 V=800.0 PL=0
MOVL C01064 V=800.0 PL=0
MOVL C01065 V=800.0 PL=0
MOVL C01066 V=800.0 PL=0
MOVL C01067 V=800.0 PL=0
MOVL C01068 V=800.0 PL=0
MOVL C01069 V=800.0 PL=0
MOVL C01070 V=800.0 PL=0
MOVL C01071 V=800.0 PL=0
MOVL C01072 V=800.0 PL=0
MOVL C01073 V=800.0 PL=0
MOVL C01074 V=800.0 PL=0
MOVL C01075 V=800.0 PL=0
MOVL C01076 V=800.0 PL=0
MOVL C01077 V=800.0 PL=0
MOVL C01078 V=800.0 PL=0
MOVL C01079 V=800.0 PL=0
MOVL C01080 V=800.0 PL=0
MOVL C01081 V=800.0 PL=0
MOVL C01082 V=800.0 PL=0
MOVL C01083 V=800.0 PL=0
MOVL C01084 V=800.0 PL=0
MOVL C01085 V=800.0 PL=0
MOVL C01086 V=800.0 PL=0
MOVL C01087 V=800.0 PL=0
MOVL C01088 V=800.0 PL=0
MOVL C01089 V=800.0 PL=0
MOVL C01090 V=800.0 PL=0
MOVL C01091 V=800.0 PL=0
MOVL C01092 V=800.0 PL=0
MOVL C01093 V=800.0 PL=0
MOVL C01094 V=800.0 PL=0
MOVL C01095 V=800.0 PL=0
MOVL C01096 V=800.0 PL=0
MOVL C01097 V=800.0 PL=0
MOVL C01098 V=800.0 PL=0
MOVL C01099 V=800.0 PL=0
MOVL C01100 V=800.0 PL=0
MOVL C01101 V=800.0 PL=0
MOVL C01102 V=800.0 PL=0
MOVL C01103 V=800.0 PL=0
MOVL C01104 V=800.0 PL=0
MOVL C01105 V=800.0 PL=0
MOVL C01106 V=800.0 PL=0
MOVL C01107 V=800.0 PL=0
MOVL C01108 V=800.0 PL=0
MOVL C01109 V=800.0 PL=0
MOVL C01110 V=800.0 PL=0
MOVL C01111 V=800.0 PL=0
MOVL C01112 V=800.0 PL=0
MOVL C01113 V=800.0 PL=0
MOVL C01114 V=800.0 PL=0
MOVL C01115 V=800.0 PL=0
MOVL C01116 V=800.0 PL=0
MOVL C01117 V=800.0 PL=0
MOVL C01118 V=800.0 PL=0
MOVL C01119 V=800.0 PL=0
MOVL C01120 V=800.0 PL=0
MOVL C01121 V=800.0 PL=0
MOVL C01122 V=800.0 PL=0
MOVL C01123 V=800.0 PL=0
MOVL C01124 V=800.0 PL=0
MOVL C01125 V=800.0 PL=0
MOVL C01126 V=800.0 PL=0
MOVL C01127 V=800.0 PL=0
MOVL C01128 V=800.0 PL=0
MOVL C01129 V=800.0 PL=0
MOVL C01130 V=800.0 PL=0
MOVL C01131 V=800.0 PL=0
MOVL C01132 V=800.0 PL=0
MOVL C01133 V=800.0 PL=0
MOVL C01134 V=800.0 PL=0
MOVL C01135 V=800.0 PL=0
MOVL C01136 V=800.0 PL=0
MOVL C01137 V=800.0 PL=0
MOVL C01138 V=800.0 PL=0
MOVL C01139 V=800.0 PL=0
MOVL C01140 V=800.0 PL=0
MOVL C01141 V=800.0 PL=0
MOVL C01142 V=800.0 PL=0
MOVL C01143 V=800.0 PL=0
MOVL C01144 V=800.0 PL=0
MOVL C01145 V=800.0 PL=0
MOVL C01146 V=800.0 PL=0
MOVL C01147 V=800.0 PL=0
MOVL C01148 V=800.0 PL=0
MOVL C01149 V=800.0 PL=0
MOVL C01150 V=800.0 PL=0
MOVL C01151 V=800.0 PL=0
MOVL C01152 V=800.0 PL=0
MOVL C01153 V=800.0 PL=0
MOVL C01154 V=800.0 PL=0
MOVL C01155 V=800.0 PL=0
MOVL C01156 V=800.0 PL=0
MOVL C01157 V=800.0 PL=0
MOVL C01158 V=800.0 PL=0
MOVL C01159 V=800.0 PL=0
MOVL C01160 V=800.0 PL=0
MOVL C01161 V=800.0 PL=0
MOVL C01162 V=800.0 PL=0
MOVL C01163 V=800.0 PL=0
MOVL C01164 V=800.0 PL=0
MOVL C01165 V=800.0 PL=0
MOVL C01166 V=800.0 PL=0
MOVL C01167 V=800.0 PL=0
MOVL C01168 V=800.0 PL=0
MOVL C01169 V=800.0 PL=0
MOVL C01170 V=800.0 PL=0
MOVL C01171 V=800.0 PL=0
MOVL C01172 V=800.0 PL=0
MOVL C01173 V=800.0 PL=0
MOVL C01174 V=800.0 PL=0
MOVL C01175 V=800.0 PL=0
MOVL C01176 V=800.0 PL=0
MOVL C01177 V=800.0 PL=0
MOVL C01178 V=800.0 PL=0
MOVL C01179 V=800.0 PL=0
MOVL C01180 V=800.0 PL=0
MOVL C01181 V=800.0 PL=0
MOVL C01182 V=800.0 PL=0
MOVL C01183 V=800.0 PL=0
MOVL C01184 V=800.0 PL=0
MOVL C01185 V=800.0 PL=0
MOVL C01186 V=800.0 PL=0
MOVL C01187 V=800.0 PL=0
MOVL C01188 V=800.0 PL=0
MOVL C01189 V=800.0 PL=0
MOVL C01190 V=800.0 PL=0
MOVL C01191 V=800.0 PL=0
MOVL C01192 V=800.0 PL=0
MOVL C01193 V=800.0 PL=0
MOVL C01194 V=800.0 PL=0
MOVL C01195 V=800.0 PL=0
MOVL C01196 V=800.0 PL=0
MOVL C01197 V=800.0 PL=0
MOVL C01198 V=800.0 PL=0
MOVL C01199 V=800.0 PL=0
MOVL C01200 V=800.0 PL=0
MOVL C01201 V=800.0 PL=0
MOVL C01202 V=800.0 PL=0
MOVL C01203 V=800.0 PL=0
MOVL C01204 V=800.0 PL=0
MOVL C01205 V=800.0 PL=0
MOVL C01206 V=800.0 PL=0
MOVL C01207 V=800.0 PL=0
MOVL C01208 V=800.0 PL=0
MOVL C01209 V=800.0 PL=0
MOVL C01210 V=800.0 PL=0
MOVL C01211 V=800.0 PL=0
MOVL C01212 V=800.0 PL=0
MOVL C01213 V=800.0 PL=0
MOVL C01214 V=800.0 PL=0
MOVL C01215 V=800.0 PL=0
MOVL C01216 V=800.0 PL=0
MOVL C01217 V=800.0 PL=0
MOVL C01218 V=800.0 PL=0
MOVL C01219 V=800.0 PL=0
MOVL C01220 V=800.0 PL=0
MOVL C01221 V=800.0 PL=0
MOVL C01222 V=800.0 PL=0
MOVL C01223 V=800.0 PL=0
MOVL C01224 V=800.0 PL=0
MOVL C01225 V=800.0 PL=0
MOVL C01226 V=800.0 PL=0
MOVL C01227 V=800.0 PL=0
MOVL C01228 V=800.0 PL=0
MOVL C01229 V=800.0 PL=0
MOVL C01230 V=800.0 PL=0
MOVL C01231 V=800.0 PL=0
MOVL C01232 V=800.0 PL=0
MOVL C01233 V=800.0 PL=0
MOVL C01234 V=800.0 PL=0
MOVL C01235 V=800.0 PL=0
MOVL C01236 V=800.0 PL=0
MOVL C01237 V=800.0 PL=0
MOVL C01238 V=800.0 PL=0
MOVL C01239 V=800.0 PL=0
MOVL C01240 V=800.0 PL=0
MOVL C01241 V=800.0 PL=0
MOVL C01242 V=800.0 PL=0
MOVL C01243 V=800.0 PL=0
MOVL C01244 V=800.0 PL=0
MOVL C01245 V=800.0 PL=0
MOVL C01246 V=800.0 PL=0
MOVL C01247 V=800.0 PL=0
MOVL C01248 V=800.0 PL=0
MOVL C01249 V=800.0 PL=0
MOVL C01250 V=800.0 PL=0
MOVL C01251 V=800.0 PL=0
MOVL C01252 V=800.0 PL=0
MOVL C01253 V=800.0 PL=0
MOVL C01254 V=800.0 PL=0
MOVL C01255 V=800.0 PL=0
MOVL C01256 V=800.0 PL=0
MOVL C01257 V=800.0 PL=0
MOVL C01258 V=800.0 PL=0
MOVL C01259 V=800.0 PL=0
MOVL C01260 V=800.0 PL=0
MOVL C01261 V=800.0 PL=0
MOVL C01262 V=800.0 PL=0
MOVL C01263 V=800.0 PL=0
MOVL C01264 V=800.0 PL=0
MOVL C01265 V=800.0 PL=0
MOVL C01266 V=800.0 PL=0
MOVL C01267 V=800.0 PL=0
MOVL C01268 V=800.0 PL=0
MOVL C01269 V=800.0 PL=0
MOVL C01270 V=800.0 PL=0
MOVL C01271 V=800.0 PL=0
MOVL C01272 V=800.0 PL=0
MOVL C01273 V=800.0 PL=0
MOVL C01274 V=800.0 PL=0
MOVL C01275 V=800.0 PL=0
MOVL C01276 V=800.0 PL=0
MOVL C01277 V=800.0 PL=0
MOVL C01278 V=800.0 PL=0
MOVL C01279 V=800.0 PL=0
MOVL C01280 V=800.0 PL=0
MOVL C01281 V=800.0 PL=0
MOVL C01282 V=800.0 PL=0
MOVL C01283 V=800.0 PL=0
MOVL C01284 V=800.0 PL=0
MOVL C01285 V=800.0 PL=0
MOVL C01286 V=800.0 PL=0
MOVL C01287 V=800.0 PL=0
MOVL C01288 V=800.0 PL=0
MOVL C01289 V=800.0 PL=0
MOVL C01290 V=800.0 PL=0
MOVL C01291 V=800.0 PL=0
MOVL C01292 V=800.0 PL=0
MOVL C01293 V=800.0 PL=0
MOVL C01294 V=800.0 PL=0
MOVL C01295 V=800.0 PL=0
MOVL C01296 V=800.0 PL=0
MOVL C01297 V=800.0 PL=0
MOVL C01298 V=800.0 PL=0
MOVL C01299 V=800.0 PL=0
MOVL C01300 V=800.0 PL=0
MOVL C01301 V=800.0 PL=0
MOVL C01302 V=800.0 PL=0
MOVL C01303 V=800.0 PL=0
MOVL C01304 V=800.0 PL=0
MOVL C01305 V=800.0 PL=0
MOVL C01306 V=800.0 PL=0
MOVL C01307 V=800.0 PL=0
MOVL C01308 V=800.0 PL=0
MOVL C01309 V=800.0 PL=0
MOVL C01310 V=800.0 PL=0
MOVL C01311 V=800.0 PL=0
MOVL C01312 V=800.0 PL=0
MOVL C01313 V=800.0 PL=0
MOVL C01314 V=800.0 PL=0
MOVL C01315 V=800.0 PL=0
MOVL C01316 V=800.0 PL=0
MOVL C01317 V=800.0 PL=0
MOVL C01318 V=800.0 PL=0
MOVL C01319 V=800.0 PL=0
MOVL C01320 V=800.0 PL=0
MOVL C01321 V=800.0 PL=0
MOVL C01322 V=800.0 PL=0
MOVL C01323 V=800.0 PL=0
MOVL C01324 V=800.0 PL=0
MOVL C01325 V=800.0 PL=0
MOVL C01326 V=800.0 PL=0
MOVL C01327 V=800.0 PL=0
MOVL C01328 V=800.0 PL=0
MOVL C01329 V=800.0 PL=0
MOVL C01330 V=800.0 PL=0
MOVL C01331 V=800.0 PL=0
MOVL C01332 V=800.0 PL=0
MOVL C01333 V=800.0 PL=0
MOVL C01334 V=800.0 PL=0
MOVL C01335 V=800.0 PL=0
MOVL C01336 V=800.0 PL=0
MOVL C01337 V=800.0 PL=0
MOVL C01338 V=800.0 PL=0
MOVL C01339 V=800.0 PL=0
MOVL C01340 V=800.0 PL=0
MOVL C01341 V=800.0 PL=0
MOVL C01342 V=800.0 PL=0
MOVL C01343 V=800.0 PL=0
MOVL C01344 V=800.0 PL=0
MOVL C01345 V=800.0 PL=0
MOVL C01346 V=800.0 PL=0
MOVL C01347 V=800.0 PL=0
MOVL C01348 V=800.0 PL=0
MOVL C01349 V=800.0 PL=0
MOVL C01350 V=800.0 PL=0
MOVL C01351 V=800.0 PL=0
MOVL C01352 V=800.0 PL=0
MOVL C01353 V=800.0 PL=0
MOVL C01354 V=800.0 PL=0
MOVL C01355 V=800.0 PL=0
MOVL C01356 V=800.0 PL=0
MOVL C01357 V=800.0 PL=0
MOVL C01358 V=800.0 PL=0
MOVL C01359 V=800.0 PL=0
MOVL C01360 V=800.0 PL=0
MOVL C01361 V=800.0 PL=0
MOVL C01362 V=800.0 PL=0
MOVL C01363 V=800.0 PL=0
MOVL C01364 V=800.0 PL=0
MOVL C01365 V=800.0 PL=0
MOVL C01366 V=800.0 PL=0
MOVL C01367 V=800.0 PL=0
MOVL C01368 V=800.0 PL=0
MOVL C01369 V=800.0 PL=0
MOVL C01370 V=800.0 PL=0
MOVL C01371 V=800.0 PL=0
MOVL C01372 V=800.0 PL=0
MOVL C01373 V=800.0 PL=0
MOVL C01374 V=800.0 PL=0
MOVL C01375 V=800.0 PL=0
MOVL C01376 V=800.0 PL=0
MOVL C01377 V=800.0 PL=0
MOVL C01378 V=800.0 PL=0
MOVL C01379 V=800.0 PL=0
MOVL C01380 V=800.0 PL=0
MOVL C01381 V=800.0 PL=0
MOVL C01382 V=800.0 PL=0
MOVL C01383 V=800.0 PL=0
MOVL C01384 V=800.0 PL=0
MOVL C01385 V=800.0 PL=0
MOVL C01386 V=800.0 PL=0
MOVL C01387 V=800.0 PL=0
MOVL C01388 V=800.0 PL=0
MOVL C01389 V=800.0 PL=0
MOVL C01390 V=800.0 PL=0
MOVL C01391 V=800.0 PL=0
MOVL C01392 V=800.0 PL=0
MOVL C01393 V=800.0 PL=0
MOVL C01394 V=800.0 PL=0
MOVL C01395 V=800.0 PL=0
MOVL C01396 V=800.0 PL=0
MOVL C01397 V=800.0 PL=0
MOVL C01398 V=800.0 PL=0
MOVL C01399 V=800.0 PL=0
MOVL C01400 V=800.0 PL=0
MOVL C01401 V=800.0 PL=0
MOVL C01402 V=800.0 PL=0
MOVL C01403 V=800.0 PL=0
MOVL C01404 V=800.0 PL=0
MOVL C01405 V=800.0 PL=0
MOVL C01406 V=800.0 PL=0
MOVL C01407 V=800.0 PL=0
MOVL C01408 V=800.0 PL=0
MOVL C01409 V=800.0 PL=0
MOVL C01410 V=800.0 PL=0
MOVL C01411 V=800.0 PL=0
MOVL C01412 V=800.0 PL=0
MOVL C01413 V=800.0 PL=0
MOVL C01414 V=800.0 PL=0
MOVL C01415 V=800.0 PL=0
MOVL C01416 V=800.0 PL=0
MOVL C01417 V=800.0 PL=0
MOVL C01418 V=800.0 PL=0
MOVL C01419 V=800.0 PL=0
MOVL C01420 V=800.0 PL=0
MOVL C01421 V=800.0 PL=0
MOVL C01422 V=800.0 PL=0
MOVL C01423 V=800.0 PL=0
MOVL C01424 V=800.0 PL=0
MOVL C01425 V=800.0 PL=0
MOVL C01426 V=800.0 PL=0
MOVL C01427 V=800.0 PL=0
MOVL C01428 V=800.0 PL=0
MOVL C01429 V=800.0 PL=0
MOVL C01430 V=800.0 PL=0
MOVL C01431 V=800.0 PL=0
MOVL C01432 V=800.0 PL=0
MOVL C01433 V=800.0 PL=0
MOVL C01434 V=800.0 PL=0
MOVL C01435 V=800.0 PL=0
MOVL C01436 V=800.0 PL=0
MOVL C01437 V=800.0 PL=0
MOVL C01438 V=800.0 PL=0
MOVL C01439 V=800.0 PL=0
MOVL C01440 V=800.0 PL=0
MOVL C01441 V=800.0 PL=0
MOVL C01442 V=800.0 PL=0
MOVL C01443 V=800.0 PL=0
MOVL C01444 V=800.0 PL=0
MOVL C01445 V=800.0 PL=0
MOVL C01446 V=800.0 PL=0
MOVL C01447 V=800.0 PL=0
MOVL C01448 V=800.0 PL=0
MOVL C01449 V=800.0 PL=0
MOVL C01450 V=800.0 PL=0
MOVL C01451 V=800.0 PL=0
MOVL C01452 V=800.0 PL=0
MOVL C01453 V=800.0 PL=0
MOVL C01454 V=800.0 PL=0
MOVL C01455 V=800.0 PL=0
MOVL C01456 V=800.0 PL=0
MOVL C01457 V=800.0 PL=0
MOVL C01458 V=800.0 PL=0
MOVL C01459 V=800.0 PL=0
MOVL C01460 V=800.0 PL=0
MOVL C01461 V=800.0 PL=0
MOVL C01462 V=800.0 PL=0
MOVL C01463 V=800.0 PL=0
MOVL C01464 V=800.0 PL=0
MOVL C01465 V=800.0 PL=0
MOVL C01466 V=800.0 PL=0
MOVL C01467 V=800.0 PL=0
MOVL C01468 V=800.0 PL=0
MOVL C01469 V=800.0 PL=0
MOVL C01470 V=800.0 PL=0
MOVL C01471 V=800.0 PL=0
MOVL C01472 V=800.0 PL=0
MOVL C01473 V=800.0 PL=0
MOVL C01474 V=800.0 PL=0
MOVL C01475 V=800.0 PL=0
MOVL C01476 V=800.0 PL=0
MOVL C01477 V=800.0 PL=0
MOVL C01478 V=800.0 PL=0
MOVL C01479 V=800.0 PL=0
MOVL C01480 V=800.0 PL=0
MOVL C01481 V=800.0 PL=0
MOVL C01482 V=800.0 PL=0
MOVL C01483 V=800.0 PL=0
MOVL C01484 V=800.0 PL=0
MOVL C01485 V=800.0 PL=0
MOVL C01486 V=800.0 PL=0
MOVL C01487 V=800.0 PL=0
MOVL C01488 V=800.0 PL=0
MOVL C01489 V=800.0 PL=0
MOVL C01490 V=800.0 PL=0
MOVL C01491 V=800.0 PL=0
MOVL C01492 V=800.0 PL=0
MOVL C01493 V=800.0 PL=0
MOVL C01494 V=800.0 PL=0
MOVL C01495 V=800.0 PL=0
MOVL C01496 V=800.0 PL=0
MOVL C01497 V=800.0 PL=0
MOVL C01498 V=800.0 PL=0
MOVL C01499 V=800.0 PL=0
MOVL C01500 V=800.0 PL=0
MOVL C01501 V=800.0 PL=0
MOVL C01502 V=800.0 PL=0
MOVL C01503 V=800.0 PL=0
MOVL C01504 V=800.0 PL=0
MOVL C01505 V=800.0 PL=0
MOVL C01506 V=800.0 PL=0
MOVL C01507 V=800.0 PL=0
MOVL C01508 V=800.0 PL=0
MOVL C01509 V=800.0 PL=0
MOVL C01510 V=800.0 PL=0
MOVL C01511 V=800.0 PL=0
MOVL C01512 V=800.0 PL=0
MOVL C01513 V=800.0 PL=0
MOVL C01514 V=800.0 PL=0
MOVL C01515 V=800.0 PL=0
MOVL C01516 V=800.0 PL=0
MOVL C01517 V=800.0 PL=0
MOVL C01518 V=800.0 PL=0
MOVL C01519 V=800.0 PL=0
MOVL C01520 V=800.0 PL=0
MOVL C01521 V=800.0 PL=0
MOVL C01522 V=800.0 PL=0
MOVL C01523 V=800.0 PL=0
MOVL C01524 V=800.0 PL=0
MOVL C01525 V=800.0 PL=0
MOVL C01526 V=800.0 PL=0
MOVL C01527 V=800.0 PL=0
MOVL C01528 V=800.0 PL=0
MOVL C01529 V=800.0 PL=0
MOVL C01530 V=800.0 PL=0
MOVL C01531 V=800.0 PL=0
MOVL C01532 V=800.0 PL=0
MOVL C01533 V=800.0 PL=0
MOVL C01534 V=800.0 PL=0
MOVL C01535 V=800.0 PL=0
MOVL C01536 V=800.0 PL=0
MOVL C01537 V=800.0 PL=0
MOVL C01538 V=800.0 PL=0
MOVL C01539 V=800.0 PL=0
MOVL C01540 V=800.0 PL=0
MOVL C01541 V=800.0 PL=0
MOVL C01542 V=800.0 PL=0
MOVL C01543 V=800.0 PL=0
MOVL C01544 V=800.0 PL=0
MOVL C01545 V=800.0 PL=0
MOVL C01546 V=800.0 PL=0
MOVL C01547 V=800.0 PL=0
MOVL C01548 V=800.0 PL=0
MOVL C01549 V=800.0 PL=0
MOVL C01550 V=800.0 PL=0
MOVL C01551 V=800.0 PL=0
MOVL C01552 V=800.0 PL=0
MOVL C01553 V=800.0 PL=0
MOVL C01554 V=800.0 PL=0
MOVL C01555 V=800.0 PL=0
MOVL C01556 V=800.0 PL=0
MOVL C01557 V=800.0 PL=0
MOVL C01558 V=800.0 PL=0
MOVL C01559 V=800.0 PL=0
MOVL C01560 V=800.0 PL=0
MOVL C01561 V=800.0 PL=0
MOVL C01562 V=800.0 PL=0
MOVL C01563 V=800.0 PL=0
MOVL C01564 V=800.0 PL=0
MOVL C01565 V=800.0 PL=0
MOVL C01566 V=800.0 PL=0
MOVL C01567 V=800.0 PL=0
MOVL C01568 V=800.0 PL=0
MOVL C01569 V=800.0 PL=0
MOVL C01570 V=800.0 PL=0
MOVL C01571 V=800.0 PL=0
MOVL C01572 V=800.0 PL=0
MOVL C01573 V=800.0 PL=0
MOVL C01574 V=800.0 PL=0
MOVL C01575 V=800.0 PL=0
MOVL C01576 V=800.0 PL=0
MOVL C01577 V=800.0 PL=0
MOVL C01578 V=800.0 PL=0
MOVL C01579 V=800.0 PL=0
MOVL C01580 V=800.0 PL=0
MOVL C01581 V=800.0 PL=0
MOVL C01582 V=800.0 PL=0
MOVL C01583 V=800.0 PL=0
MOVL C01584 V=800.0 PL=0
MOVL C01585 V=800.0 PL=0
MOVL C01586 V=800.0 PL=0
MOVL C01587 V=800.0 PL=0
MOVL C01588 V=800.0 PL=0
MOVL C01589 V=800.0 PL=0
MOVL C01590 V=800.0 PL=0
MOVL C01591 V=800.0 PL=0
MOVL C01592 V=800.0 PL=0
MOVL C01593 V=800.0 PL=0
MOVL C01594 V=800.0 PL=0
MOVL C01595 V=800.0 PL=0
MOVL C01596 V=800.0 PL=0
MOVL C01597 V=800.0 PL=0
MOVL C01598 V=800.0 PL=0
MOVL C01599 V=800.0 PL=0
MOVL C01600 V=800.0 PL=0
MOVL C01601 V=800.0 PL=0
MOVL C01602 V=800.0 PL=0
MOVL C01603 V=800.0 PL=0
MOVL C01604 V=800.0 PL=0
MOVL C01605 V=800.0 PL=0
MOVL C01606 V=800.0 PL=0
MOVL C01607 V=800.0 PL=0
MOVL C01608 V=800.0 PL=0
MOVL C01609 V=800.0 PL=0
MOVL C01610 V=800.0 PL=0
MOVL C01611 V=800.0 PL=0
MOVL C01612 V=800.0 PL=0
MOVL C01613 V=800.0 PL=0
MOVL C01614 V=800.0 PL=0
MOVL C01615 V=800.0 PL=0
MOVL C01616 V=800.0 PL=0
MOVL C01617 V=800.0 PL=0
MOVL C01618 V=800.0 PL=0
MOVL C01619 V=800.0 PL=0
MOVL C01620 V=800.0 PL=0
MOVL C01621 V=800.0 PL=0
MOVL C01622 V=800.0 PL=0
MOVL C01623 V=800.0 PL=0
MOVL C01624 V=800.0 PL=0
MOVL C01625 V=800.0 PL=0
MOVL C01626 V=800.0 PL=0
MOVL C01627 V=800.0 PL=0
MOVL C01628 V=800.0 PL=0
MOVL C01629 V=800.0 PL=0
MOVL C01630 V=800.0 PL=0
MOVL C01631 V=800.0 PL=0
MOVL C01632 V=800.0 PL=0
MOVL C01633 V=800.0 PL=0
MOVL C01634 V=800.0 PL=0
MOVL C01635 V=800.0 PL=0
MOVL C01636 V=800.0 PL=0
MOVL C01637 V=800.0 PL=0
MOVL C01638 V=800.0 PL=0
MOVL C01639 V=800.0 PL=0
MOVL C01640 V=800.0 PL=0
MOVL C01641 V=800.0 PL=0
MOVL C01642 V=800.0 PL=0
MOVL C01643 V=800.0 PL=0
MOVL C01644 V=800.0 PL=0
MOVL C01645 V=800.0 PL=0
MOVL C01646 V=800.0 PL=0
MOVL C01647 V=800.0 PL=0
MOVL C01648 V=800.0 PL=0
MOVL C01649 V=800.0 PL=0
MOVL C01650 V=800.0 PL=0
MOVL C01651 V=800.0 PL=0
MOVL C01652 V=800.0 PL=0
MOVL C01653 V=800.0 PL=0
MOVL C01654 V=800.0 PL=0
MOVL C01655 V=800.0 PL=0
MOVL C01656 V=800.0 PL=0
MOVL C01657 V=800.0 PL=0
MOVL C01658 V=800.0 PL=0
MOVL C01659 V=800.0 PL=0
MOVL C01660 V=800.0 PL=0
MOVL C01661 V=800.0 PL=0
MOVL C01662 V=800.0 PL=0
MOVL C01663 V=800.0 PL=0
MOVL C01664 V=800.0 PL=0
MOVL C01665 V=800.0 PL=0
MOVL C01666 V=800.0 PL=0
MOVL C01667 V=800.0 PL=0
MOVL C01668 V=800.0 PL=0
MOVL C01669 V=800.0 PL=0
MOVL C01670 V=800.0 PL=0
MOVL C01671 V=800.0 PL=0
MOVL C01672 V=800.0 PL=0
MOVL C01673 V=800.0 PL=0
MOVL C01674 V=800.0 PL=0
MOVL C01675 V=800.0 PL=0
MOVL C01676 V=800.0 PL=0
MOVL C01677 V=800.0 PL=0
MOVL C01678 V=800.0 PL=0
MOVL C01679 V=800.0 PL=0
MOVL C01680 V=800.0 PL=0
MOVL C01681 V=800.0 PL=0
MOVL C01682 V=800.0 PL=0
MOVL C01683 V=800.0 PL=0
MOVL C01684 V=800.0 PL=0
MOVL C01685 V=800.0 PL=0
MOVL C01686 V=800.0 PL=0
MOVL C01687 V=800.0 PL=0
MOVL C01688 V=800.0 PL=0
MOVL C01689 V=800.0 PL=0
MOVL C01690 V=800.0 PL=0
MOVL C01691 V=800.0 PL=0
MOVL C01692 V=800.0 PL=0
MOVL C01693 V=800.0 PL=0
MOVL C01694 V=800.0 PL=0
MOVL C01695 V=800.0 PL=0
MOVL C01696 V=800.0 PL=0
MOVL C01697 V=800.0 PL=0
MOVL C01698 V=800.0 PL=0
MOVL C01699 V=800.0 PL=0
MOVL C01700 V=800.0 PL=0
MOVL C01701 V=800.0 PL=0
MOVL C01702 V=800.0 PL=0
MOVL C01703 V=800.0 PL=0
MOVL C01704 V=800.0 PL=0
MOVL C01705 V=800.0 PL=0
MOVL C01706 V=800.0 PL=0
MOVL C01707 V=800.0 PL=0
MOVL C01708 V=800.0 PL=0
MOVL C01709 V=800.0 PL=0
MOVL C01710 V=800.0 PL=0
MOVL C01711 V=800.0 PL=0
MOVL C01712 V=800.0 PL=0
MOVL C01713 V=800.0 PL=0
MOVL C01714 V=800.0 PL=0
MOVL C01715 V=800.0 PL=0
MOVL C01716 V=800.0 PL=0
MOVL C01717 V=800.0 PL=0
MOVL C01718 V=800.0 PL=0
MOVL C01719 V=800.0 PL=0
MOVL C01720 V=800.0 PL=0
MOVL C01721 V=800.0 PL=0
MOVL C01722 V=800.0 PL=0
MOVL C01723 V=800.0 PL=0
MOVL C01724 V=800.0 PL=0
MOVL C01725 V=800.0 PL=0
MOVL C01726 V=800.0 PL=0
MOVL C01727 V=800.0 PL=0
MOVL C01728 V=800.0 PL=0
MOVL C01729 V=800.0 PL=0
MOVL C01730 V=800.0 PL=0
MOVL C01731 V=800.0 PL=0
MOVL C01732 V=800.0 PL=0
MOVL C01733 V=800.0 PL=0
MOVL C01734 V=800.0 PL=0
MOVL C01735 V=800.0 PL=0
MOVL C01736 V=800.0 PL=0
MOVL C01737 V=800.0 PL=0
MOVL C01738 V=800.0 PL=0
MOVL C01739 V=800.0 PL=0
MOVL C01740 V=800.0 PL=0
MOVL C01741 V=800.0 PL=0
MOVL C01742 V=800.0 PL=0
MOVL C01743 V=800.0 PL=0
MOVL C01744 V=800.0 PL=0
MOVL C01745 V=800.0 PL=0
MOVL C01746 V=800.0 PL=0
MOVL C01747 V=800.0 PL=0
MOVL C01748 V=800.0 PL=0
MOVL C01749 V=800.0 PL=0
MOVL C01750 V=800.0 PL=0
MOVL C01751 V=800.0 PL=0
MOVL C01752 V=800.0 PL=0
MOVL C01753 V=800.0 PL=0
MOVL C01754 V=800.0 PL=0
MOVL C01755 V=800.0 PL=0
MOVL C01756 V=800.0 PL=0
MOVL C01757 V=800.0 PL=0
MOVL C01758 V=800.0 PL=0
MOVL C01759 V=800.0 PL=0
MOVL C01760 V=800.0 PL=0
MOVL C01761 V=800.0 PL=0
MOVL C01762 V=800.0 PL=0
MOVL C01763 V=800.0 PL=0
MOVL C01764 V=800.0 PL=0
MOVL C01765 V=800.0 PL=0
MOVL C01766 V=800.0 PL=0
MOVL C01767 V=800.0 PL=0
MOVL C01768 V=800.0 PL=0
MOVL C01769 V=800.0 PL=0
MOVL C01770 V=800.0 PL=0
MOVL C01771 V=800.0 PL=0
MOVL C01772 V=800.0 PL=0
MOVL C01773 V=800.0 PL=0
MOVL C01774 V=800.0 PL=0
MOVL C01775 V=800.0 PL=0
MOVL C01776 V=800.0 PL=0
MOVL C01777 V=800.0 PL=0
MOVL C01778 V=800.0 PL=0
MOVL C01779 V=800.0 PL=0
MOVL C01780 V=800.0 PL=0
MOVL C01781 V=800.0 PL=0
MOVL C01782 V=800.0 PL=0
MOVL C01783 V=800.0 PL=0
MOVL C01784 V=800.0 PL=0
MOVL C01785 V=800.0 PL=0
MOVL C01786 V=800.0 PL=0
MOVL C01787 V=800.0 PL=0
MOVL C01788 V=800.0 PL=0
MOVL C01789 V=800.0 PL=0
MOVL C01790 V=800.0 PL=0
MOVL C01791 V=800.0 PL=0
MOVL C01792 V=800.0 PL=0
MOVL C01793 V=800.0 PL=0
MOVL C01794 V=800.0 PL=0
MOVL C01795 V=800.0 PL=0
MOVL C01796 V=800.0 PL=0
MOVL C01797 V=800.0 PL=0
MOVL C01798 V=800.0 PL=0
MOVL C01799 V=800.0 PL=0
MOVL C01800 V=800.0 PL=0
MOVL C01801 V=800.0 PL=0
MOVL C01802 V=800.0 PL=0
MOVL C01803 V=800.0 PL=0
MOVL C01804 V=800.0 PL=0
MOVL C01805 V=800.0 PL=0
MOVL C01806 V=800.0 PL=0
MOVL C01807 V=800.0 PL=0
MOVL C01808 V=800.0 PL=0
MOVL C01809 V=800.0 PL=0
MOVL C01810 V=800.0 PL=0
MOVL C01811 V=800.0 PL=0
MOVL C01812 V=800.0 PL=0
MOVL C01813 V=800.0 PL=0
MOVL C01814 V=800.0 PL=0
MOVL C01815 V=800.0 PL=0
MOVL C01816 V=800.0 PL=0
MOVL C01817 V=800.0 PL=0
MOVL C01818 V=800.0 PL=0
MOVL C01819 V=800.0 PL=0
MOVL C01820 V=800.0 PL=0
MOVL C01821 V=800.0 PL=0
MOVL C01822 V=800.0 PL=0
MOVL C01823 V=800.0 PL=0
MOVL C01824 V=800.0 PL=0
MOVL C01825 V=800.0 PL=0
MOVL C01826 V=800.0 PL=0
MOVL C01827 V=800.0 PL=0
MOVL C01828 V=800.0 PL=0
MOVL C01829 V=800.0 PL=0
MOVL C01830 V=800.0 PL=0
MOVL C01831 V=800.0 PL=0
MOVL C01832 V=800.0 PL=0
MOVL C01833 V=800.0 PL=0
MOVL C01834 V=800.0 PL=0
MOVL C01835 V=800.0 PL=0
MOVL C01836 V=800.0 PL=0
MOVL C01837 V=800.0 PL=0
MOVL C01838 V=800.0 PL=0
MOVL C01839 V=800.0 PL=0
MOVL C01840 V=800.0 PL=0
MOVL C01841 V=800.0 PL=0
MOVL C01842 V=800.0 PL=0
MOVL C01843 V=800.0 PL=0
MOVL C01844 V=800.0 PL=0
MOVL C01845 V=800.0 PL=0
MOVL C01846 V=800.0 PL=0
MOVL C01847 V=800.0 PL=0
MOVL C01848 V=800.0 PL=0
MOVL C01849 V=800.0 PL=0
MOVL C01850 V=800.0 PL=0
MOVL C01851 V=800.0 PL=0
MOVL C01852 V=800.0 PL=0
MOVL C01853 V=800.0 PL=0
MOVL C01854 V=800.0 PL=0
MOVL C01855 V=800.0 PL=0
MOVL C01856 V=800.0 PL=0
MOVL C01857 V=800.0 PL=0
MOVL C01858 V=800.0 PL=0
MOVL C01859 V=800.0 PL=0
MOVL C01860 V=800.0 PL=0
MOVL C01861 V=800.0 PL=0
MOVL C01862 V=800.0 PL=0
MOVL C01863 V=800.0 PL=0
MOVL C01864 V=800.0 PL=0
MOVL C01865 V=800.0 PL=0
MOVL C01866 V=800.0 PL=0
MOVL C01867 V=800.0 PL=0
MOVL C01868 V=800.0 PL=0
MOVL C01869 V=800.0 PL=0
MOVL C01870 V=800.0 PL=0
MOVL C01871 V=800.0 PL=0
MOVL C01872 V=800.0 PL=0
MOVL C01873 V=800.0 PL=0
MOVL C01874 V=800.0 PL=0
MOVL C01875 V=800.0 PL=0
MOVL C01876 V=800.0 PL=0
MOVL C01877 V=800.0 PL=0
MOVL C01878 V=800.0 PL=0
MOVL C01879 V=800.0 PL=0
MOVL C01880 V=800.0 PL=0
MOVL C01881 V=800.0 PL=0
MOVL C01882 V=800.0 PL=0
MOVL C01883 V=800.0 PL=0
MOVL C01884 V=800.0 PL=0
MOVL C01885 V=800.0 PL=0
MOVL C01886 V=800.0 PL=0
MOVL C01887 V=800.0 PL=0
MOVL C01888 V=800.0 PL=0
MOVL C01889 V=800.0 PL=0
MOVL C01890 V=800.0 PL=0
MOVL C01891 V=800.0 PL=0
MOVL C01892 V=800.0 PL=0
MOVL C01893 V=800.0 PL=0
MOVL C01894 V=800.0 PL=0
MOVL C01895 V=800.0 PL=0
MOVL C01896 V=800.0 PL=0
MOVL C01897 V=800.0 PL=0
MOVL C01898 V=800.0 PL=0
MOVL C01899 V=800.0 PL=0
MOVL C01900 V=800.0 PL=0
MOVL C01901 V=800.0 PL=0
MOVL C01902 V=800.0 PL=0
MOVL C01903 V=800.0 PL=0
MOVL C01904 V=800.0 PL=0
MOVL C01905 V=800.0 PL=0
MOVL C01906 V=800.0 PL=0
MOVL C01907 V=800.0 PL=0
MOVL C01908 V=800.0 PL=0
MOVL C01909 V=800.0 PL=0
MOVL C01910 V=800.0 PL=0
MOVL C01911 V=800.0 PL=0
MOVL C01912 V=800.0 PL=0
MOVL C01913 V=800.0 PL=0
MOVL C01914 V=800.0 PL=0
MOVL C01915 V=800.0 PL=0
MOVL C01916 V=800.0 PL=0
MOVL C01917 V=800.0 PL=0
MOVL C01918 V=800.0 PL=0
MOVL C01919 V=800.0 PL=0
MOVL C01920 V=800.0 PL=0
MOVL C01921 V=800.0 PL=0
MOVL C01922 V=800.0 PL=0
MOVL C01923 V=800.0 PL=0
MOVL C01924 V=800.0 PL=0
MOVL C01925 V=800.0 PL=0
MOVL C01926 V=800.0 PL=0
MOVL C01927 V=800.0 PL=0
MOVL C01928 V=800.0 PL=0
MOVL C01929 V=800.0 PL=0
MOVL C01930 V=800.0 PL=0
MOVL C01931 V=800.0 PL=0
MOVL C01932 V=800.0 PL=0
MOVL C01933 V=800.0 PL=0
MOVL C01934 V=800.0 PL=0
MOVL C01935 V=800.0 PL=0
MOVL C01936 V=800.0 PL=0
MOVL C01937 V=800.0 PL=0
MOVL C01938 V=800.0 PL=0
MOVL C01939 V=800.0 PL=0
MOVL C01940 V=800.0 PL=0
MOVL C01941 V=800.0 PL=0
MOVL C01942 V=800.0 PL=0
MOVL C01943 V=800.0 PL=0
MOVL C01944 V=800.0 PL=0
MOVL C01945 V=800.0 PL=0
MOVL C01946 V=800.0 PL=0
MOVL C01947 V=800.0 PL=0
MOVL C01948 V=800.0 PL=0
MOVL C01949 V=800.0 PL=0
MOVL C01950 V=800.0 PL=0
MOVL C01951 V=800.0 PL=0
MOVL C01952 V=800.0 PL=0
MOVL C01953 V=800.0 PL=0
MOVL C01954 V=800.0 PL=0
MOVL C01955 V=800.0 PL=0
MOVL C01956 V=800.0 PL=0
MOVL C01957 V=800.0 PL=0
MOVL C01958 V=800.0 PL=0
MOVL C01959 V=800.0 PL=0
MOVL C01960 V=800.0 PL=0
MOVL C01961 V=800.0 PL=0
MOVL C01962 V=800.0 PL=0
MOVL C01963 V=800.0 PL=0
MOVL C01964 V=800.0 PL=0
MOVL C01965 V=800.0 PL=0
MOVL C01966 V=800.0 PL=0
MOVL C01967 V=800.0 PL=0
MOVL C01968 V=800.0 PL=0
MOVL C01969 V=800.0 PL=0
MOVL C01970 V=800.0 PL=0
MOVL C01971 V=800.0 PL=0
MOVL C01972 V=800.0 PL=0
MOVL C01973 V=800.0 PL=0
MOVL C01974 V=800.0 PL=0
MOVL C01975 V=800.0 PL=0
MOVL C01976 V=800.0 PL=0
MOVL C01977 V=800.0 PL=0
MOVL C01978 V=800.0 PL=0
MOVL C01979 V=800.0 PL=0
MOVL C01980 V=800.0 PL=0
MOVL C01981 V=800.0 PL=0
MOVL C01982 V=800.0 PL=0
MOVL C01983 V=800.0 PL=0
MOVL C01984 V=800.0 PL=0
MOVL C01985 V=800.0 PL=0
MOVL C01986 V=800.0 PL=0
MOVL C01987 V=800.0 PL=0
MOVL C01988 V=800.0 PL=0
MOVL C01989 V=800.0 PL=0
MOVL C01990 V=800.0 PL=0
MOVL C01991 V=800.0 PL=0
MOVL C01992 V=800.0 PL=0
MOVL C01993 V=800.0 PL=0
MOVL C01994 V=800.0 PL=0
MOVL C01995 V=800.0 PL=0
MOVL C01996 V=800.0 PL=0
MOVL C01997 V=800.0 PL=0
MOVL C01998 V=800.0 PL=0
MOVL C01999 V=800.0 PL=0
MOVL C02000 V=800.0 PL=0
MOVL C02001 V=800.0 PL=0
MOVL C02002 V=800.0 PL=0
MOVL C02003 V=800.0 PL=0
MOVL C02004 V=800.0 PL=0
MOVL C02005 V=800.0 PL=0
MOVL C02006 V=800.0 PL=0
MOVL C02007 V=800.0 PL=0
MOVL C02008 V=800.0 PL=0
MOVL C02009 V=800.0 PL=0
MOVL C02010 V=800.0 PL=0
MOVL C02011 V=800.0 PL=0
MOVL C02012 V=800.0 PL=0
MOVL C02013 V=800.0 PL=0
MOVL C02014 V=800.0 PL=0
MOVL C02015 V=800.0 PL=0
MOVL C02016 V=800.0 PL=0
MOVL C02017 V=800.0 PL=0
MOVL C02018 V=800.0 PL=0
MOVL C02019 V=800.0 PL=0
MOVL C02020 V=800.0 PL=0
MOVL C02021 V=800.0 PL=0
MOVL C02022 V=800.0 PL=0
MOVL C02023 V=800.0 PL=0
MOVL C02024 V=800.0 PL=0
MOVL C02025 V=800.0 PL=0
MOVL C02026 V=800.0 PL=0
MOVL C02027 V=800.0 PL=0
MOVL C02028 V=800.0 PL=0
MOVL C02029 V=800.0 PL=0
MOVL C02030 V=800.0 PL=0
MOVL C02031 V=800.0 PL=0
MOVL C02032 V=800.0 PL=0
MOVL C02033 V=800.0 PL=0
MOVL C02034 V=800.0 PL=0
MOVL C02035 V=800.0 PL=0
MOVL C02036 V=800.0 PL=0
MOVL C02037 V=800.0 PL=0
MOVL C02038 V=800.0 PL=0
MOVL C02039 V=800.0 PL=0
MOVL C02040 V=800.0 PL=0
MOVL C02041 V=800.0 PL=0
MOVL C02042 V=800.0 PL=0
MOVL C02043 V=800.0 PL=0
MOVL C02044 V=800.0 PL=0
MOVL C02045 V=800.0 PL=0
MOVL C02046 V=800.0 PL=0
MOVL C02047 V=800.0 PL=0
MOVL C02048 V=800.0 PL=0
MOVL C02049 V=800.0 PL=0
MOVL C02050 V=800.0 PL=0
MOVL C02051 V=800.0 PL=0
MOVL C02052 V=800.0 PL=0
MOVL C02053 V=800.0 PL=0
MOVL C02054 V=800.0 PL=0
MOVL C02055 V=800.0 PL=0
MOVL C02056 V=800.0 PL=0
MOVL C02057 V=800.0 PL=0
MOVL C02058 V=800.0 PL=0
MOVL C02059 V=800.0 PL=0
MOVL C02060 V=800.0 PL=0
MOVL C02061 V=800.0 PL=0
MOVL C02062 V=800.0 PL=0
MOVL C02063 V=800.0 PL=0
MOVL C02064 V=800.0 PL=0
MOVL C02065 V=800.0 PL=0
MOVL C02066 V=800.0 PL=0
MOVL C02067 V=800.0 PL=0
MOVL C02068 V=800.0 PL=0
MOVL C02069 V=800.0 PL=0
MOVL C02070 V=800.0 PL=0
MOVL C02071 V=800.0 PL=0
MOVL C02072 V=800.0 PL=0
MOVL C02073 V=800.0 PL=0
MOVL C02074 V=800.0 PL=0
MOVL C02075 V=800.0 PL=0
MOVL C02076 V=800.0 PL=0
MOVL C02077 V=800.0 PL=0
MOVL C02078 V=800.0 PL=0
MOVL C02079 V=800.0 PL=0
MOVL C02080 V=800.0 PL=0
MOVL C02081 V=800.0 PL=0
MOVL C02082 V=800.0 PL=0
MOVL C02083 V=800.0 PL=0
MOVL C02084 V=800.0 PL=0
MOVL C02085 V=800.0 PL=0
MOVL C02086 V=800.0 PL=0
